LIN {X 0,Y 185.248,Z 515.043,A -85,B 0,C 180,E1 -23455.315,E2 -23455.315} C_VEL
LIN {X 0,Y 180.266,Z 523.701,A -85,B 0,C 180,E1 -23458.243,E2 -23458.243} C_VEL
LIN {X 0,Y 175.893,Z 530.639,A -85,B 0,C 180,E1 -23461.349,E2 -23461.349} C_VEL
LIN {X 0,Y 172.117,Z 536.223,A -85,B 0,C 180,E1 -23464.612,E2 -23464.612} C_VEL
LIN {X 0,Y 168.809,Z 540.646,A -85,B 0,C 180,E1 -23467.994,E2 -23467.994} C_VEL
LIN {X 0,Y 166.906,Z 542.994,A -85,B 0,C 180,E1 -23470.314,E2 -23470.314} C_VEL
LIN {X 0,Y 165.318,Z 544.923,A -85,B 0,C 180,E1 -23472.687,E2 -23472.687} C_VEL
LIN {X 0,Y 164.124,Z 546.443,A -85,B 0,C 180,E1 -23475.112,E2 -23475.112} C_VEL
LIN {X 0,Y 162.456,Z 548.229,A -85,B 0,C 180,E1 -23480.035,E2 -23480.035} C_VEL
LIN {X 0,Y 161.851,Z 548.504,A -85,B 0,C 180,E1 -23485.017,E2 -23485.017} C_VEL
LIN {X 0,Y 161.843,Z 548.032,A -85,B 0,C 180,E1 -23487.511,E2 -23487.511} C_VEL
LIN {X 0,Y 161.944,Z 547.156,A -85,B 0,C 180,E1 -23490,E2 -23490} C_VEL
LIN {X 0,Y 161.834,Z 545.704,A -85,B 0,C 180,E1 -23492.768,E2 -23492.768} C_VEL
LIN {X 0,Y 161.908,Z 543.109,A -85,B 0,C 180,E1 -23496.229,E2 -23496.229} C_VEL
LIN {X 0,Y 162.4,Z 539.305,A -85,B 0,C 180,E1 -23499.968,E2 -23499.968} C_VEL
LIN {X 0,Y 163.325,Z 534.348,A -85,B 0,C 180,E1 -23503.689,E2 -23503.689} C_VEL
LIN {X 0,Y 164.915,Z 528.1,A -85,B 0,C 180,E1 -23507.355,E2 -23507.355} C_VEL
LIN {X 0,Y 167.043,Z 520.275,A -85,B 0,C 180,E1 -23510.953,E2 -23510.953} C_VEL
LIN {X 0,Y 168.207,Z 515.825,A -85,B 0,C 180,E1 -23512.657,E2 -23512.657} C_VEL
LIN {X 0,Y 170.737,Z 506.615,A -85,B 0,C 180,E1 -23515.607,E2 -23515.607} C_VEL
LIN {X 0,Y 172.299,Z 500.233,A -85,B 0,C 180,E1 -23517.314,E2 -23517.314} C_VEL
LIN {X 0,Y 172.549,Z 488.695,A -85,B 0,C 180,E1 -23520.136,E2 -23520.136} C_VEL
LIN {X 0,Y 171.858,Z 483.921,A -85,B 0,C 180,E1 -23521.271,E2 -23521.271} C_VEL
LIN {X 0,Y 168.91,Z 476.415,A -85,B 0,C 180,E1 -23523.212,E2 -23523.212} C_VEL
LIN {X 0,Y 166.129,Z 470.335,A -85,B 0,C 180,E1 -23524.727,E2 -23524.727} C_VEL
LIN {X 0,Y 164.489,Z 465.427,A -85,B 0,C 180,E1 -23525.769,E2 -23525.769} C_VEL
LIN {X 0,Y 164.105,Z 463.69,A -85,B 0,C 180,E1 -23526.084,E2 -23526.084} C_VEL
LIN {X 0,Y 161.974,Z 452.52,A -85,B 0,C 180,E1 -23527.886,E2 -23527.886} C_VEL
LIN {X 0,Y 160.13,Z 446.258,A -85,B 0,C 180,E1 -23528.883,E2 -23528.883} C_VEL
LIN {X 0,Y 158.77,Z 443.265,A -85,B 0,C 180,E1 -23529.445,E2 -23529.445} C_VEL
LIN {X 0,Y 158.538,Z 442.036,A -85,B 0,C 180,E1 -23529.667,E2 -23529.667} C_VEL
LIN {X 0,Y 157.914,Z 438.937,A -85,B 0,C 180,E1 -23534.594,E2 -23534.594} C_VEL
LIN {X 0,Y 157.284,Z 435.898,A -85,B 0,C 180,E1 -23539.983,E2 -23539.983} C_VEL
LIN {X 0,Y 157.277,Z 435.896,A -85,B 0,C 180,E1 -23544.485,E2 -23544.485} C_VEL
LIN {X 0,Y 157.29,Z 435.892,A -85,B 0,C 180,E1 -23548.095,E2 -23548.095} C_VEL
LIN {X 0,Y 157.319,Z 435.868,A -85,B 0,C 180,E1 -23553.465,E2 -23553.465} C_VEL
LIN {X 0,Y 157.391,Z 435.873,A -85,B 0,C 180,E1 -23559.667,E2 -23559.667} C_VEL
LIN {X 0,Y 157.436,Z 435.841,A -85,B 0,C 180,E1 -23564.464,E2 -23564.464} C_VEL
LIN {X 0,Y 157.744,Z 435.835,A -85,B 0,C 180,E1 -23569.734,E2 -23569.734} C_VEL
LIN {X 0,Y 157.816,Z 435.818,A -85,B 0,C 180,E1 -23572.322,E2 -23572.322} C_VEL
LIN {X 0,Y 158.255,Z 435.755,A -85,B 0,C 180,E1 -23580,E2 -23580} C_VEL
LIN {X 0,Y 157.807,Z 435.813,A -85,B 0,C 180,E1 -23587.678,E2 -23587.678} C_VEL
LIN {X 0,Y 157.668,Z 435.803,A -85,B 0,C 180,E1 -23591.301,E2 -23591.301} C_VEL
LIN {X 0,Y 157.45,Z 435.863,A -85,B 0,C 180,E1 -23595.534,E2 -23595.534} C_VEL
LIN {X 0,Y 157.366,Z 435.877,A -85,B 0,C 180,E1 -23600.933,E2 -23600.933} C_VEL
LIN {X 0,Y 157.306,Z 435.888,A -85,B 0,C 180,E1 -23606.681,E2 -23606.681} C_VEL
LIN {X 0,Y 157.273,Z 435.894,A -85,B 0,C 180,E1 -23612.427,E2 -23612.427} C_VEL
LIN {X 0,Y 157.322,Z 435.881,A -85,B 0,C 180,E1 -23616.478,E2 -23616.478} C_VEL
LIN {X 0,Y 157.293,Z 435.891,A -85,B 0,C 180,E1 -23622.083,E2 -23622.083} C_VEL
LIN {X 0,Y 157.311,Z 435.889,A -85,B 0,C 180,E1 -23625.627,E2 -23625.627} C_VEL
LIN {X 0,Y 157.29,Z 435.892,A -85,B 0,C 180,E1 -23631.279,E2 -23631.279} C_VEL
LIN {X 0,Y 157.293,Z 435.89,A -85,B 0,C 180,E1 -23634.491,E2 -23634.491} C_VEL
LIN {X 0,Y 157.293,Z 435.892,A -85,B 0,C 180,E1 -23638.096,E2 -23638.096} C_VEL
LIN {X 0,Y 157.413,Z 436.05,A -85,B 0,C 180,E1 -23644.324,E2 -23644.324} C_VEL
LIN {X 0,Y 158.472,Z 438.848,A -85,B 0,C 180,E1 -23644.818,E2 -23644.818} C_VEL
LIN {X 0,Y 159.937,Z 441.308,A -85,B 0,C 180,E1 -23645.373,E2 -23645.373} C_VEL
LIN {X 0,Y 162.244,Z 447.436,A -85,B 0,C 180,E1 -23646.537,E2 -23646.537} C_VEL
LIN {X 0,Y 165.121,Z 458.356,A -85,B 0,C 180,E1 -23648.593,E2 -23648.593} C_VEL
LIN {X 0,Y 166.934,Z 469.095,A -85,B 0,C 180,E1 -23650.769,E2 -23650.769} C_VEL
LIN {X 0,Y 167.973,Z 478.773,A -85,B 0,C 180,E1 -23652.97,E2 -23652.97} C_VEL
LIN {X 0,Y 168.048,Z 485.349,A -85,B 0,C 180,E1 -23654.587,E2 -23654.587} C_VEL
LIN {X 0,Y 165.391,Z 495.531,A -85,B 0,C 180,E1 -23657.11,E2 -23657.11} C_VEL
LIN {X 0,Y 162.736,Z 504.865,A -85,B 0,C 180,E1 -23660.053,E2 -23660.053} C_VEL
LIN {X 0,Y 160.012,Z 513.909,A -85,B 0,C 180,E1 -23663.697,E2 -23663.697} C_VEL
LIN {X 0,Y 157.857,Z 521.199,A -85,B 0,C 180,E1 -23667.449,E2 -23667.449} C_VEL
LIN {X 0,Y 156.377,Z 527.011,A -85,B 0,C 180,E1 -23671.288,E2 -23671.288} C_VEL
LIN {X 0,Y 155.326,Z 531.874,A -85,B 0,C 180,E1 -23675.485,E2 -23675.485} C_VEL
LIN {X 0,Y 154.858,Z 534.018,A -85,B 0,C 180,E1 -23677.826,E2 -23677.826} C_VEL
LIN {X 0,Y 154.489,Z 536.015,A -85,B 0,C 180,E1 -23680.485,E2 -23680.485} C_VEL
LIN {X 0,Y 154.366,Z 537.581,A -85,B 0,C 180,E1 -23683.158,E2 -23683.158} C_VEL
LIN {X 0,Y 154.602,Z 539.136,A -85,B 0,C 180,E1 -23687.327,E2 -23687.327} C_VEL
LIN {X 0,Y 155.216,Z 539.674,A -85,B 0,C 180,E1 -23691.237,E2 -23691.237} C_VEL
LIN {X 0,Y 156.841,Z 539.037,A -85,B 0,C 180,E1 -23696.339,E2 -23696.339} C_VEL
LIN {X 0,Y 158.206,Z 537.971,A -85,B 0,C 180,E1 -23699.252,E2 -23699.252} C_VEL
LIN {X 0,Y 159.765,Z 536.553,A -85,B 0,C 180,E1 -23701.862,E2 -23701.862} C_VEL
LIN {X 0,Y 162.668,Z 533.529,A -85,B 0,C 180,E1 -23705.68,E2 -23705.68} C_VEL
LIN {X 0,Y 166.199,Z 529.371,A -85,B 0,C 180,E1 -23709.368,E2 -23709.368} C_VEL
LIN {X 0,Y 170.381,Z 523.946,A -85,B 0,C 180,E1 -23712.89,E2 -23712.89} C_VEL
LIN {X 0,Y 175.179,Z 517.076,A -85,B 0,C 180,E1 -23716.231,E2 -23716.231} C_VEL
LIN {X 0,Y 180.487,Z 508.46,A -85,B 0,C 180,E1 -23719.403,E2 -23719.403} C_VEL
LIN {X 0,Y 182.402,Z 505.098,A -85,B 0,C 180,E1 -23720.408,E2 -23720.408} C_VEL
LIN {X 0,Y 183.047,Z 501.795,A -85,B 0,C 180,E1 -23721.655,E2 -23721.655} C_VEL
LIN {X 0,Y 183.419,Z 493.353,A -85,B 0,C 180,E1 -23724.918,E2 -23724.918} C_VEL
LIN {X 0,Y 182.864,Z 486.054,A -85,B 0,C 180,E1 -23727.727,E2 -23727.727} C_VEL
LIN {X 0,Y 181.46,Z 479.589,A -85,B 0,C 180,E1 -23730.426,E2 -23730.426} C_VEL
LIN {X 0,Y 178.98,Z 472.271,A -85,B 0,C 180,E1 -23733.785,E2 -23733.785} C_VEL
LIN {X 0,Y 177.584,Z 468.714,A -85,B 0,C 180,E1 -23735.537,E2 -23735.537} C_VEL
LIN {X 0,Y 175.789,Z 464.643,A -85,B 0,C 180,E1 -23737.679,E2 -23737.679} C_VEL
LIN {X 0,Y 172.805,Z 459.443,A -85,B 0,C 180,E1 -23741.013,E2 -23741.013} C_VEL
LIN {X 0,Y 170.994,Z 455.9,A -85,B 0,C 180,E1 -23743.28,E2 -23743.28} C_VEL
LIN {X 0,Y 168.006,Z 451.559,A -85,B 0,C 180,E1 -23747.007,E2 -23747.007} C_VEL
LIN {X 0,Y 167.308,Z 449.863,A -85,B 0,C 180,E1 -23748.184,E2 -23748.184} C_VEL
LIN {X 0,Y 164.416,Z 446.661,A -85,B 0,C 180,E1 -23752.478,E2 -23752.478} C_VEL
LIN {X 0,Y 163.46,Z 444.35,A -85,B 0,C 180,E1 -23754.758,E2 -23754.758} C_VEL
LIN {X 0,Y 161.309,Z 442.705,A -85,B 0,C 180,E1 -23760,E2 -23760} C_VEL
LIN {X 0,Y 160.22,Z 442.45,A -85,B 0,C 180,E1 -23767.562,E2 -23767.562} C_VEL
LIN {X 0,Y 160.844,Z 443.769,A -85,B 0,C 180,E1 -23772.62,E2 -23772.62} C_VEL
LIN {X 0,Y 163.558,Z 446.46,A -85,B 0,C 180,E1 -23779.484,E2 -23779.484} C_VEL
LIN {X 0,Y 164.954,Z 450.06,A -85,B 0,C 180,E1 -23782.548,E2 -23782.548} C_VEL
LIN {X 0,Y 167.772,Z 453.476,A -85,B 0,C 180,E1 -23786.429,E2 -23786.429} C_VEL
LIN {X 0,Y 169.173,Z 456.816,A -85,B 0,C 180,E1 -23788.539,E2 -23788.539} C_VEL
LIN {X 0,Y 171.221,Z 459.675,A -85,B 0,C 180,E1 -23790.868,E2 -23790.868} C_VEL
LIN {X 0,Y 172.912,Z 463.461,A -85,B 0,C 180,E1 -23792.999,E2 -23792.999} C_VEL
LIN {X 0,Y 174.138,Z 465.815,A -85,B 0,C 180,E1 -23794.404,E2 -23794.404} C_VEL
LIN {X 0,Y 176.569,Z 471.344,A -85,B 0,C 180,E1 -23797.245,E2 -23797.245} C_VEL
LIN {X 0,Y 179.659,Z 479.366,A -85,B 0,C 180,E1 -23800.938,E2 -23800.938} C_VEL
LIN {X 0,Y 181.699,Z 487.258,A -85,B 0,C 180,E1 -23804.126,E2 -23804.126} C_VEL
LIN {X 0,Y 182.158,Z 491.421,A -85,B 0,C 180,E1 -23805.602,E2 -23805.602} C_VEL
LIN {X 0,Y 182.082,Z 499.048,A -85,B 0,C 180,E1 -23808.149,E2 -23808.149} C_VEL
LIN {X 0,Y 180.895,Z 508.937,A -85,B 0,C 180,E1 -23811.566,E2 -23811.566} C_VEL
LIN {X 0,Y 179.382,Z 515.508,A -85,B 0,C 180,E1 -23814.007,E2 -23814.007} C_VEL
LIN {X 0,Y 175.101,Z 522.707,A -85,B 0,C 180,E1 -23816.504,E2 -23816.504} C_VEL
LIN {X 0,Y 170.424,Z 529.828,A -85,B 0,C 180,E1 -23819.658,E2 -23819.658} C_VEL
LIN {X 0,Y 165.735,Z 536.348,A -85,B 0,C 180,E1 -23823.561,E2 -23823.561} C_VEL
LIN {X 0,Y 162.222,Z 540.694,A -85,B 0,C 180,E1 -23827.051,E2 -23827.051} C_VEL
LIN {X 0,Y 158.529,Z 544.901,A -85,B 0,C 180,E1 -23831.921,E2 -23831.921} C_VEL
LIN {X 0,Y 157.231,Z 546.355,A -85,B 0,C 180,E1 -23834.443,E2 -23834.443} C_VEL
LIN {X 0,Y 155.456,Z 548.072,A -85,B 0,C 180,E1 -23839.581,E2 -23839.581} C_VEL
LIN {X 0,Y 154.76,Z 548.267,A -85,B 0,C 180,E1 -23844.789,E2 -23844.789} C_VEL
LIN {X 0,Y 154.758,Z 547.701,A -85,B 0,C 180,E1 -23847.558,E2 -23847.558} C_VEL
LIN {X 0,Y 154.854,Z 546.841,A -85,B 0,C 180,E1 -23849.999,E2 -23849.999} C_VEL
LIN {X 0,Y 154.742,Z 545.519,A -85,B 0,C 180,E1 -23852.603,E2 -23852.603} C_VEL
LIN {X 0,Y 154.855,Z 542.694,A -85,B 0,C 180,E1 -23856.514,E2 -23856.514} C_VEL
LIN {X 0,Y 155.4,Z 538.819,A -85,B 0,C 180,E1 -23860.421,E2 -23860.421} C_VEL
LIN {X 0,Y 156.397,Z 533.783,A -85,B 0,C 180,E1 -23864.308,E2 -23864.308} C_VEL
LIN {X 0,Y 158.11,Z 527.447,A -85,B 0,C 180,E1 -23868.128,E2 -23868.128} C_VEL
LIN {X 0,Y 160.414,Z 519.48,A -85,B 0,C 180,E1 -23871.863,E2 -23871.863} C_VEL
LIN {X 0,Y 162.42,Z 512.051,A -85,B 0,C 180,E1 -23874.675,E2 -23874.675} C_VEL
LIN {X 0,Y 165.153,Z 502.458,A -85,B 0,C 180,E1 -23877.565,E2 -23877.565} C_VEL
LIN {X 0,Y 165.664,Z 497.782,A -85,B 0,C 180,E1 -23878.852,E2 -23878.852} C_VEL
LIN {X 0,Y 165.875,Z 487.286,A -85,B 0,C 180,E1 -23881.466,E2 -23881.466} C_VEL
LIN {X 0,Y 165.536,Z 476.278,A -85,B 0,C 180,E1 -23883.79,E2 -23883.79} C_VEL
LIN {X 0,Y 164.288,Z 464.832,A -85,B 0,C 180,E1 -23885.892,E2 -23885.892} C_VEL
LIN {X 0,Y 164.105,Z 463.69,A -85,B 0,C 180,E1 -23886.084,E2 -23886.084} C_VEL
LIN {X 0,Y 162.955,Z 460.45,A -85,B 0,C 180,E1 -23886.762,E2 -23886.762} C_VEL
LIN {X 0,Y 159.595,Z 455.978,A -85,B 0,C 180,E1 -23888.04,E2 -23888.04} C_VEL
LIN {X 0,Y 155.141,Z 450.752,A -85,B 0,C 180,E1 -23889.646,E2 -23889.646} C_VEL
LIN {X 0,Y 153.972,Z 448.703,A -85,B 0,C 180,E1 -23890.138,E2 -23890.138} C_VEL
LIN {X 0,Y 152.57,Z 445.411,A -85,B 0,C 180,E1 -23890.784,E2 -23890.784} C_VEL
LIN {X 0,Y 151.417,Z 442.505,A -85,B 0,C 180,E1 -23891.333,E2 -23891.333} C_VEL
LIN {X 0,Y 151.297,Z 441.796,A -85,B 0,C 180,E1 -23891.519,E2 -23891.519} C_VEL
LIN {X 0,Y 150.741,Z 439.381,A -85,B 0,C 180,E1 -23895.625,E2 -23895.625} C_VEL
LIN {X 0,Y 150.224,Z 436.778,A -85,B 0,C 180,E1 -23900.399,E2 -23900.399} C_VEL
LIN {X 0,Y 150.188,Z 436.777,A -85,B 0,C 180,E1 -23905.837,E2 -23905.837} C_VEL
LIN {X 0,Y 150.204,Z 436.771,A -85,B 0,C 180,E1 -23909.023,E2 -23909.023} C_VEL
LIN {X 0,Y 150.241,Z 436.745,A -85,B 0,C 180,E1 -23912.717,E2 -23912.717} C_VEL
LIN {X 0,Y 150.348,Z 436.752,A -85,B 0,C 180,E1 -23919.207,E2 -23919.207} C_VEL
LIN {X 0,Y 150.346,Z 436.72,A -85,B 0,C 180,E1 -23923.711,E2 -23923.711} C_VEL
LIN {X 0,Y 150.658,Z 436.718,A -85,B 0,C 180,E1 -23929.245,E2 -23929.245} C_VEL
LIN {X 0,Y 150.752,Z 436.701,A -85,B 0,C 180,E1 -23931.96,E2 -23931.96} C_VEL
LIN {X 0,Y 151.215,Z 436.631,A -85,B 0,C 180,E1 -23940,E2 -23940} C_VEL
LIN {X 0,Y 150.741,Z 436.689,A -85,B 0,C 180,E1 -23948.04,E2 -23948.04} C_VEL
LIN {X 0,Y 150.602,Z 436.681,A -85,B 0,C 180,E1 -23951.491,E2 -23951.491} C_VEL
LIN {X 0,Y 150.358,Z 436.749,A -85,B 0,C 180,E1 -23956.287,E2 -23956.287} C_VEL
LIN {X 0,Y 150.347,Z 436.752,A -85,B 0,C 180,E1 -23960.792,E2 -23960.792} C_VEL
LIN {X 0,Y 150.238,Z 436.767,A -85,B 0,C 180,E1 -23967.28,E2 -23967.28} C_VEL
LIN {X 0,Y 150.214,Z 436.773,A -85,B 0,C 180,E1 -23972.634,E2 -23972.634} C_VEL
LIN {X 0,Y 150.233,Z 436.767,A -85,B 0,C 180,E1 -23977.455,E2 -23977.455} C_VEL
LIN {X 0,Y 150.234,Z 436.771,A -85,B 0,C 180,E1 -23981.543,E2 -23981.543} C_VEL
LIN {X 0,Y 150.286,Z 436.764,A -85,B 0,C 180,E1 -23985.458,E2 -23985.458} C_VEL
LIN {X 0,Y 150.236,Z 436.769,A -85,B 0,C 180,E1 -23989.088,E2 -23989.088} C_VEL
LIN {X 0,Y 150.238,Z 436.77,A -85,B 0,C 180,E1 -23992.678,E2 -23992.678} C_VEL
LIN {X 0,Y 150.217,Z 436.773,A -85,B 0,C 180,E1 -23997.366,E2 -23997.366} C_VEL
LIN {X 0,Y 150.243,Z 436.771,A -85,B 0,C 180,E1 -24002.494,E2 -24002.494} C_VEL
LIN {X 0,Y 151.372,Z 439.8,A -85,B 0,C 180,E1 -24003.108,E2 -24003.108} C_VEL
LIN {X 0,Y 152.628,Z 441.712,A -85,B 0,C 180,E1 -24003.616,E2 -24003.616} C_VEL
LIN {X 0,Y 155.281,Z 446.867,A -85,B 0,C 180,E1 -24004.849,E2 -24004.849} C_VEL
LIN {X 0,Y 158.629,Z 458.919,A -85,B 0,C 180,E1 -24007.306,E2 -24007.306} C_VEL
LIN {X 0,Y 160.475,Z 470.171,A -85,B 0,C 180,E1 -24009.74,E2 -24009.74} C_VEL
LIN {X 0,Y 161.422,Z 480.564,A -85,B 0,C 180,E1 -24012.257,E2 -24012.257} C_VEL
LIN {X 0,Y 161.347,Z 486.487,A -85,B 0,C 180,E1 -24013.788,E2 -24013.788} C_VEL
LIN {X 0,Y 158.431,Z 496.914,A -85,B 0,C 180,E1 -24016.533,E2 -24016.533} C_VEL
LIN {X 0,Y 155.735,Z 506.012,A -85,B 0,C 180,E1 -24019.601,E2 -24019.601} C_VEL
LIN {X 0,Y 152.913,Z 514.903,A -85,B 0,C 180,E1 -24023.403,E2 -24023.403} C_VEL
LIN {X 0,Y 150.734,Z 522.021,A -85,B 0,C 180,E1 -24027.328,E2 -24027.328} C_VEL
LIN {X 0,Y 149.214,Z 527.691,A -85,B 0,C 180,E1 -24031.35,E2 -24031.35} C_VEL
LIN {X 0,Y 148.217,Z 532.161,A -85,B 0,C 180,E1 -24035.442,E2 -24035.442} C_VEL
LIN {X 0,Y 147.691,Z 534.539,A -85,B 0,C 180,E1 -24038.208,E2 -24038.208} C_VEL
LIN {X 0,Y 147.363,Z 536.487,A -85,B 0,C 180,E1 -24040.998,E2 -24040.998} C_VEL
LIN {X 0,Y 147.266,Z 537.961,A -85,B 0,C 180,E1 -24043.805,E2 -24043.805} C_VEL
LIN {X 0,Y 147.531,Z 539.324,A -85,B 0,C 180,E1 -24047.685,E2 -24047.685} C_VEL
LIN {X 0,Y 148.331,Z 539.896,A -85,B 0,C 180,E1 -24052.275,E2 -24052.275} C_VEL
LIN {X 0,Y 150.007,Z 539.268,A -85,B 0,C 180,E1 -24057.106,E2 -24057.106} C_VEL
LIN {X 0,Y 151.742,Z 538.013,A -85,B 0,C 180,E1 -24060.628,E2 -24060.628} C_VEL
LIN {X 0,Y 154.935,Z 535.114,A -85,B 0,C 180,E1 -24065.265,E2 -24065.265} C_VEL
LIN {X 0,Y 159.14,Z 530.647,A -85,B 0,C 180,E1 -24069.818,E2 -24069.818} C_VEL
LIN {X 0,Y 164.205,Z 524.591,A -85,B 0,C 180,E1 -24074.067,E2 -24074.067} C_VEL
LIN {X 0,Y 169.231,Z 517.827,A -85,B 0,C 180,E1 -24077.488,E2 -24077.488} C_VEL
LIN {X 0,Y 174.767,Z 509.35,A -85,B 0,C 180,E1 -24080.724,E2 -24080.724} C_VEL
LIN {X 0,Y 176.697,Z 506.03,A -85,B 0,C 180,E1 -24081.77,E2 -24081.77} C_VEL
LIN {X 0,Y 177.431,Z 500.168,A -85,B 0,C 180,E1 -24084.251,E2 -24084.251} C_VEL
LIN {X 0,Y 177.621,Z 492.175,A -85,B 0,C 180,E1 -24087.539,E2 -24087.539} C_VEL
LIN {X 0,Y 176.823,Z 486.029,A -85,B 0,C 180,E1 -24090.212,E2 -24090.212} C_VEL
LIN {X 0,Y 174.92,Z 478.606,A -85,B 0,C 180,E1 -24093.771,E2 -24093.771} C_VEL
LIN {X 0,Y 173.381,Z 474.2,A -85,B 0,C 180,E1 -24096.087,E2 -24096.087} C_VEL
LIN {X 0,Y 171.778,Z 470.128,A -85,B 0,C 180,E1 -24098.395,E2 -24098.395} C_VEL
LIN {X 0,Y 169.164,Z 465.061,A -85,B 0,C 180,E1 -24101.845,E2 -24101.845} C_VEL
LIN {X 0,Y 167.59,Z 461.677,A -85,B 0,C 180,E1 -24104.182,E2 -24104.182} C_VEL
LIN {X 0,Y 165.182,Z 457.75,A -85,B 0,C 180,E1 -24107.718,E2 -24107.718} C_VEL
LIN {X 0,Y 164.566,Z 456.199,A -85,B 0,C 180,E1 -24108.92,E2 -24108.92} C_VEL
LIN {X 0,Y 162.033,Z 452.791,A -85,B 0,C 180,E1 -24113.463,E2 -24113.463} C_VEL
LIN {X 0,Y 161.402,Z 451.058,A -85,B 0,C 180,E1 -24115.317,E2 -24115.317} C_VEL
LIN {X 0,Y 159.36,Z 449.483,A -85,B 0,C 180,E1 -24121.264,E2 -24121.264} C_VEL
LIN {X 0,Y 158.693,Z 449.486,A -85,B 0,C 180,E1 -24128.276,E2 -24128.276} C_VEL
LIN {X 0,Y 159.836,Z 451.546,A -85,B 0,C 180,E1 -24134.906,E2 -24134.906} C_VEL
LIN {X 0,Y 161.452,Z 453.152,A -85,B 0,C 180,E1 -24138.909,E2 -24138.909} C_VEL
LIN {X 0,Y 162.813,Z 456.916,A -85,B 0,C 180,E1 -24142.359,E2 -24142.359} C_VEL
LIN {X 0,Y 164.678,Z 459.264,A -85,B 0,C 180,E1 -24145.263,E2 -24145.263} C_VEL
LIN {X 0,Y 166.97,Z 464.198,A -85,B 0,C 180,E1 -24148.951,E2 -24148.951} C_VEL
LIN {X 0,Y 168.1,Z 466.338,A -85,B 0,C 180,E1 -24150.527,E2 -24150.527} C_VEL
LIN {X 0,Y 170.523,Z 471.909,A -85,B 0,C 180,E1 -24153.95,E2 -24153.95} C_VEL
LIN {X 0,Y 173.072,Z 478.552,A -85,B 0,C 180,E1 -24157.526,E2 -24157.526} C_VEL
LIN {X 0,Y 175.119,Z 485.035,A -85,B 0,C 180,E1 -24160.628,E2 -24160.628} C_VEL
LIN {X 0,Y 176.514,Z 491.858,A -85,B 0,C 180,E1 -24163.574,E2 -24163.574} C_VEL
LIN {X 0,Y 176.54,Z 498.862,A -85,B 0,C 180,E1 -24166.136,E2 -24166.136} C_VEL
LIN {X 0,Y 175.511,Z 507.179,A -85,B 0,C 180,E1 -24169.149,E2 -24169.149} C_VEL
LIN {X 0,Y 173.991,Z 514.433,A -85,B 0,C 180,E1 -24171.976,E2 -24171.976} C_VEL
LIN {X 0,Y 172.876,Z 517.473,A -85,B 0,C 180,E1 -24173.156,E2 -24173.156} C_VEL
LIN {X 0,Y 167.532,Z 525.542,A -85,B 0,C 180,E1 -24176.232,E2 -24176.232} C_VEL
LIN {X 0,Y 162.444,Z 532.614,A -85,B 0,C 180,E1 -24179.851,E2 -24179.851} C_VEL
LIN {X 0,Y 158.083,Z 538.031,A -85,B 0,C 180,E1 -24183.604,E2 -24183.604} C_VEL
LIN {X 0,Y 154.624,Z 541.949,A -85,B 0,C 180,E1 -24187.273,E2 -24187.273} C_VEL
LIN {X 0,Y 151.777,Z 544.865,A -85,B 0,C 180,E1 -24191.087,E2 -24191.087} C_VEL
LIN {X 0,Y 149.267,Z 547.279,A -85,B 0,C 180,E1 -24196.384,E2 -24196.384} C_VEL
LIN {X 0,Y 147.945,Z 548.175,A -85,B 0,C 180,E1 -24201.806,E2 -24201.806} C_VEL
LIN {X 0,Y 147.691,Z 548.014,A -85,B 0,C 180,E1 -24204.538,E2 -24204.538} C_VEL
LIN {X 0,Y 147.677,Z 547.252,A -85,B 0,C 180,E1 -24208.022,E2 -24208.022} C_VEL
LIN {X 0,Y 147.767,Z 546.522,A -85,B 0,C 180,E1 -24209.999,E2 -24209.999} C_VEL
LIN {X 0,Y 147.646,Z 545.166,A -85,B 0,C 180,E1 -24212.728,E2 -24212.728} C_VEL
LIN {X 0,Y 147.783,Z 542.271,A -85,B 0,C 180,E1 -24216.827,E2 -24216.827} C_VEL
LIN {X 0,Y 148.381,Z 538.321,A -85,B 0,C 180,E1 -24220.92,E2 -24220.92} C_VEL
LIN {X 0,Y 149.695,Z 532.204,A -85,B 0,C 180,E1 -24225.661,E2 -24225.661} C_VEL
LIN {X 0,Y 151.707,Z 525.503,A -85,B 0,C 180,E1 -24229.624,E2 -24229.624} C_VEL
LIN {X 0,Y 154.255,Z 517.157,A -85,B 0,C 180,E1 -24233.493,E2 -24233.493} C_VEL
LIN {X 0,Y 155.362,Z 512.973,A -85,B 0,C 180,E1 -24235.127,E2 -24235.127} C_VEL
LIN {X 0,Y 158.222,Z 503.532,A -85,B 0,C 180,E1 -24238.16,E2 -24238.16} C_VEL
LIN {X 0,Y 158.913,Z 499.006,A -85,B 0,C 180,E1 -24239.471,E2 -24239.471} C_VEL
LIN {X 0,Y 159.278,Z 487.857,A -85,B 0,C 180,E1 -24242.418,E2 -24242.418} C_VEL
LIN {X 0,Y 159.086,Z 477.591,A -85,B 0,C 180,E1 -24244.722,E2 -24244.722} C_VEL
LIN {X 0,Y 157.935,Z 465.896,A -85,B 0,C 180,E1 -24247.04,E2 -24247.04} C_VEL
LIN {X 0,Y 155.889,Z 454.167,A -85,B 0,C 180,E1 -24249.093,E2 -24249.093} C_VEL
LIN {X 0,Y 153.972,Z 448.703,A -85,B 0,C 180,E1 -24250.138,E2 -24250.138} C_VEL
LIN {X 0,Y 151.998,Z 445.869,A -85,B 0,C 180,E1 -24250.948,E2 -24250.948} C_VEL
LIN {X 0,Y 149.545,Z 443.812,A -85,B 0,C 180,E1 -24251.936,E2 -24251.936} C_VEL
LIN {X 0,Y 146.327,Z 441.924,A -85,B 0,C 180,E1 -24253.517,E2 -24253.517} C_VEL
LIN {X 0,Y 144.037,Z 440.581,A -85,B 0,C 180,E1 -24255.418,E2 -24255.418} C_VEL
LIN {X 0,Y 143.604,Z 439.995,A -85,B 0,C 180,E1 -24256.468,E2 -24256.468} C_VEL
LIN {X 0,Y 143.148,Z 437.659,A -85,B 0,C 180,E1 -24261.182,E2 -24261.182} C_VEL
LIN {X 0,Y 143.179,Z 437.651,A -85,B 0,C 180,E1 -24267.32,E2 -24267.32} C_VEL
LIN {X 0,Y 143.187,Z 437.623,A -85,B 0,C 180,E1 -24272.062,E2 -24272.062} C_VEL
LIN {X 0,Y 143.274,Z 437.634,A -85,B 0,C 180,E1 -24278.745,E2 -24278.745} C_VEL
LIN {X 0,Y 143.29,Z 437.598,A -85,B 0,C 180,E1 -24282.885,E2 -24282.885} C_VEL
LIN {X 0,Y 143.591,Z 437.597,A -85,B 0,C 180,E1 -24288.709,E2 -24288.709} C_VEL
LIN {X 0,Y 143.67,Z 437.586,A -85,B 0,C 180,E1 -24291.561,E2 -24291.561} C_VEL
LIN {X 0,Y 144.174,Z 437.506,A -85,B 0,C 180,E1 -24300,E2 -24300} C_VEL
LIN {X 0,Y 143.659,Z 437.566,A -85,B 0,C 180,E1 -24308.439,E2 -24308.439} C_VEL
LIN {X 0,Y 143.544,Z 437.559,A -85,B 0,C 180,E1 -24311.712,E2 -24311.712} C_VEL
LIN {X 0,Y 143.297,Z 437.633,A -85,B 0,C 180,E1 -24317.113,E2 -24317.113} C_VEL
LIN {X 0,Y 143.273,Z 437.63,A -85,B 0,C 180,E1 -24321.254,E2 -24321.254} C_VEL
LIN {X 0,Y 143.184,Z 437.641,A -85,B 0,C 180,E1 -24327.935,E2 -24327.935} C_VEL
LIN {X 0,Y 143.166,Z 437.65,A -85,B 0,C 180,E1 -24333.436,E2 -24333.436} C_VEL
LIN {X 0,Y 143.127,Z 437.655,A -85,B 0,C 180,E1 -24339.668,E2 -24339.668} C_VEL
LIN {X 0,Y 143.18,Z 437.648,A -85,B 0,C 180,E1 -24343.408,E2 -24343.408} C_VEL
LIN {X 0,Y 143.169,Z 437.651,A -85,B 0,C 180,E1 -24347.419,E2 -24347.419} C_VEL
LIN {X 0,Y 143.167,Z 437.65,A -85,B 0,C 180,E1 -24351.76,E2 -24351.76} C_VEL
LIN {X 0,Y 143.185,Z 437.649,A -85,B 0,C 180,E1 -24357.323,E2 -24357.323} C_VEL
LIN {X 0,Y 143.144,Z 437.774,A -85,B 0,C 180,E1 -24360.553,E2 -24360.553} C_VEL
LIN {X 0,Y 144.243,Z 440.681,A -85,B 0,C 180,E1 -24361.173,E2 -24361.173} C_VEL
LIN {X 0,Y 145.618,Z 442.737,A -85,B 0,C 180,E1 -24361.801,E2 -24361.801} C_VEL
LIN {X 0,Y 149.699,Z 450.427,A -85,B 0,C 180,E1 -24363.896,E2 -24363.896} C_VEL
LIN {X 0,Y 152.533,Z 461.393,A -85,B 0,C 180,E1 -24366.334,E2 -24366.334} C_VEL
LIN {X 0,Y 154.188,Z 472.769,A -85,B 0,C 180,E1 -24368.98,E2 -24368.98} C_VEL
LIN {X 0,Y 154.908,Z 482.352,A -85,B 0,C 180,E1 -24371.484,E2 -24371.484} C_VEL
LIN {X 0,Y 154.835,Z 487.061,A -85,B 0,C 180,E1 -24372.791,E2 -24372.791} C_VEL
LIN {X 0,Y 152.164,Z 496.271,A -85,B 0,C 180,E1 -24375.285,E2 -24375.285} C_VEL
LIN {X 0,Y 149.251,Z 505.528,A -85,B 0,C 180,E1 -24378.456,E2 -24378.456} C_VEL
LIN {X 0,Y 146.272,Z 514.53,A -85,B 0,C 180,E1 -24382.408,E2 -24382.408} C_VEL
LIN {X 0,Y 143.935,Z 521.778,A -85,B 0,C 180,E1 -24386.501,E2 -24386.501} C_VEL
LIN {X 0,Y 142.526,Z 526.659,A -85,B 0,C 180,E1 -24390.001,E2 -24390.001} C_VEL
LIN {X 0,Y 141.401,Z 531.175,A -85,B 0,C 180,E1 -24394.043,E2 -24394.043} C_VEL
LIN {X 0,Y 140.508,Z 535.063,A -85,B 0,C 180,E1 -24398.631,E2 -24398.631} C_VEL
LIN {X 0,Y 140.214,Z 536.935,A -85,B 0,C 180,E1 -24401.566,E2 -24401.566} C_VEL
LIN {X 0,Y 140.195,Z 538.337,A -85,B 0,C 180,E1 -24404.516,E2 -24404.516} C_VEL
LIN {X 0,Y 140.479,Z 539.513,A -85,B 0,C 180,E1 -24408.096,E2 -24408.096} C_VEL
LIN {X 0,Y 141.494,Z 540.086,A -85,B 0,C 180,E1 -24413.413,E2 -24413.413} C_VEL
LIN {X 0,Y 143.185,Z 539.505,A -85,B 0,C 180,E1 -24417.934,E2 -24417.934} C_VEL
LIN {X 0,Y 145.384,Z 538.028,A -85,B 0,C 180,E1 -24422.124,E2 -24422.124} C_VEL
LIN {X 0,Y 148.486,Z 535.408,A -85,B 0,C 180,E1 -24426.427,E2 -24426.427} C_VEL
LIN {X 0,Y 152.089,Z 531.904,A -85,B 0,C 180,E1 -24430.311,E2 -24430.311} C_VEL
LIN {X 0,Y 156.393,Z 527.232,A -85,B 0,C 180,E1 -24434.028,E2 -24434.028} C_VEL
LIN {X 0,Y 161.541,Z 520.961,A -85,B 0,C 180,E1 -24437.697,E2 -24437.697} C_VEL
LIN {X 0,Y 166.522,Z 514.126,A -85,B 0,C 180,E1 -24440.724,E2 -24440.724} C_VEL
LIN {X 0,Y 170.185,Z 508.666,A -85,B 0,C 180,E1 -24442.65,E2 -24442.65} C_VEL
LIN {X 0,Y 170.877,Z 506.927,A -85,B 0,C 180,E1 -24443.322,E2 -24443.322} C_VEL
LIN {X 0,Y 171.781,Z 500.013,A -85,B 0,C 180,E1 -24446.446,E2 -24446.446} C_VEL
LIN {X 0,Y 171.916,Z 493.981,A -85,B 0,C 180,E1 -24449.146,E2 -24449.146} C_VEL
LIN {X 0,Y 171.25,Z 488.417,A -85,B 0,C 180,E1 -24451.839,E2 -24451.839} C_VEL
LIN {X 0,Y 169.854,Z 482.595,A -85,B 0,C 180,E1 -24454.906,E2 -24454.906} C_VEL
LIN {X 0,Y 168.578,Z 478.569,A -85,B 0,C 180,E1 -24457.253,E2 -24457.253} C_VEL
LIN {X 0,Y 167.577,Z 475.464,A -85,B 0,C 180,E1 -24459.116,E2 -24459.116} C_VEL
LIN {X 0,Y 165.329,Z 470.535,A -85,B 0,C 180,E1 -24462.689,E2 -24462.689} C_VEL
LIN {X 0,Y 163.965,Z 467.36,A -85,B 0,C 180,E1 -24465.098,E2 -24465.098} C_VEL
LIN {X 0,Y 161.349,Z 462.252,A -85,B 0,C 180,E1 -24469.967,E2 -24469.967} C_VEL
LIN {X 0,Y 159.637,Z 459.567,A -85,B 0,C 180,E1 -24473.682,E2 -24473.682} C_VEL
LIN {X 0,Y 159.285,Z 458.378,A -85,B 0,C 180,E1 -24474.938,E2 -24474.938} C_VEL
LIN {X 0,Y 157.684,Z 456.449,A -85,B 0,C 180,E1 -24480,E2 -24480} C_VEL
LIN {X 0,Y 156.781,Z 456.138,A -85,B 0,C 180,E1 -24485.144,E2 -24485.144} C_VEL
LIN {X 0,Y 156.848,Z 456.591,A -85,B 0,C 180,E1 -24489.681,E2 -24489.681} C_VEL
LIN {X 0,Y 158.917,Z 459.496,A -85,B 0,C 180,E1 -24498.034,E2 -24498.034} C_VEL
LIN {X 0,Y 160.151,Z 463.362,A -85,B 0,C 180,E1 -24501.902,E2 -24501.902} C_VEL
LIN {X 0,Y 161.553,Z 465.287,A -85,B 0,C 180,E1 -24504.41,E2 -24504.41} C_VEL
LIN {X 0,Y 164.329,Z 471.511,A -85,B 0,C 180,E1 -24509.462,E2 -24509.462} C_VEL
LIN {X 0,Y 166.509,Z 477.414,A -85,B 0,C 180,E1 -24513.279,E2 -24513.279} C_VEL
LIN {X 0,Y 168.746,Z 484.184,A -85,B 0,C 180,E1 -24517.152,E2 -24517.152} C_VEL
LIN {X 0,Y 170.337,Z 490.674,A -85,B 0,C 180,E1 -24520.428,E2 -24520.428} C_VEL
LIN {X 0,Y 171.087,Z 495.532,A -85,B 0,C 180,E1 -24522.671,E2 -24522.671} C_VEL
LIN {X 0,Y 170.835,Z 501.465,A -85,B 0,C 180,E1 -24525.021,E2 -24525.021} C_VEL
LIN {X 0,Y 169.467,Z 509.814,A -85,B 0,C 180,E1 -24528.287,E2 -24528.287} C_VEL
LIN {X 0,Y 167.739,Z 516.468,A -85,B 0,C 180,E1 -24531.062,E2 -24531.062} C_VEL
LIN {X 0,Y 166.342,Z 519.376,A -85,B 0,C 180,E1 -24532.221,E2 -24532.221} C_VEL
LIN {X 0,Y 160.802,Z 527.03,A -85,B 0,C 180,E1 -24535.377,E2 -24535.377} C_VEL
LIN {X 0,Y 155.606,Z 533.676,A -85,B 0,C 180,E1 -24539.11,E2 -24539.11} C_VEL
LIN {X 0,Y 150.434,Z 539.547,A -85,B 0,C 180,E1 -24543.652,E2 -24543.652} C_VEL
LIN {X 0,Y 146.999,Z 543.035,A -85,B 0,C 180,E1 -24547.513,E2 -24547.513} C_VEL
LIN {X 0,Y 145.065,Z 544.812,A -85,B 0,C 180,E1 -24550.176,E2 -24550.176} C_VEL
LIN {X 0,Y 142.343,Z 547.156,A -85,B 0,C 180,E1 -24555.707,E2 -24555.707} C_VEL
LIN {X 0,Y 140.908,Z 547.965,A -85,B 0,C 180,E1 -24561.394,E2 -24561.394} C_VEL
LIN {X 0,Y 140.587,Z 547.176,A -85,B 0,C 180,E1 -24567.134,E2 -24567.134} C_VEL
LIN {X 0,Y 140.69,Z 546.204,A -85,B 0,C 180,E1 -24569.999,E2 -24569.999} C_VEL
LIN {X 0,Y 140.55,Z 544.797,A -85,B 0,C 180,E1 -24572.866,E2 -24572.866} C_VEL
LIN {X 0,Y 140.738,Z 541.843,A -85,B 0,C 180,E1 -24577.171,E2 -24577.171} C_VEL
LIN {X 0,Y 141.384,Z 537.817,A -85,B 0,C 180,E1 -24581.468,E2 -24581.468} C_VEL
LIN {X 0,Y 142.831,Z 531.583,A -85,B 0,C 180,E1 -24586.434,E2 -24586.434} C_VEL
LIN {X 0,Y 144.996,Z 524.79,A -85,B 0,C 180,E1 -24590.572,E2 -24590.572} C_VEL
LIN {X 0,Y 147.636,Z 516.307,A -85,B 0,C 180,E1 -24594.615,E2 -24594.615} C_VEL
LIN {X 0,Y 150.051,Z 508.728,A -85,B 0,C 180,E1 -24597.469,E2 -24597.469} C_VEL
LIN {X 0,Y 152.049,Z 501.324,A -85,B 0,C 180,E1 -24599.793,E2 -24599.793} C_VEL
LIN {X 0,Y 152.637,Z 491.163,A -85,B 0,C 180,E1 -24602.751,E2 -24602.751} C_VEL
LIN {X 0,Y 152.762,Z 481.673,A -85,B 0,C 180,E1 -24605.102,E2 -24605.102} C_VEL
LIN {X 0,Y 152.066,Z 471.097,A -85,B 0,C 180,E1 -24607.435,E2 -24607.435} C_VEL
LIN {X 0,Y 150.577,Z 459.871,A -85,B 0,C 180,E1 -24609.635,E2 -24609.635} C_VEL
LIN {X 0,Y 149.017,Z 453.455,A -85,B 0,C 180,E1 -24610.88,E2 -24610.88} C_VEL
LIN {X 0,Y 145.626,Z 445.665,A -85,B 0,C 180,E1 -24612.649,E2 -24612.649} C_VEL
LIN {X 0,Y 144.149,Z 442.365,A -85,B 0,C 180,E1 -24613.39,E2 -24613.39} C_VEL
LIN {X 0,Y 143.989,Z 441.577,A -85,B 0,C 180,E1 -24613.558,E2 -24613.558} C_VEL
LIN {X 0,Y 143.604,Z 439.995,A -85,B 0,C 180,E1 -24616.468,E2 -24616.468} C_VEL
LIN {X 0,Y 142.753,Z 439.046,A -85,B 0,C 180,E1 -24618.764,E2 -24618.764} C_VEL
LIN {X 0,Y 141.063,Z 438.573,A -85,B 0,C 180,E1 -24621.05,E2 -24621.05} C_VEL
LIN {X 0,Y 136.404,Z 438.516,A -85,B 0,C 180,E1 -24627.398,E2 -24627.398} C_VEL
LIN {X 0,Y 136.054,Z 438.531,A -85,B 0,C 180,E1 -24629.08,E2 -24629.08} C_VEL
LIN {X 0,Y 136.144,Z 438.499,A -85,B 0,C 180,E1 -24632.315,E2 -24632.315} C_VEL
LIN {X 0,Y 136.241,Z 438.51,A -85,B 0,C 180,E1 -24638.832,E2 -24638.832} C_VEL
LIN {X 0,Y 136.262,Z 438.478,A -85,B 0,C 180,E1 -24645.055,E2 -24645.055} C_VEL
LIN {X 0,Y 136.494,Z 438.478,A -85,B 0,C 180,E1 -24648.114,E2 -24648.114} C_VEL
LIN {X 0,Y 136.595,Z 438.467,A -85,B 0,C 180,E1 -24651.12,E2 -24651.12} C_VEL
LIN {X 0,Y 137.131,Z 438.381,A -85,B 0,C 180,E1 -24659.999,E2 -24659.999} C_VEL
LIN {X 0,Y 136.587,Z 438.439,A -85,B 0,C 180,E1 -24668.879,E2 -24668.879} C_VEL
LIN {X 0,Y 136.488,Z 438.437,A -85,B 0,C 180,E1 -24671.954,E2 -24671.954} C_VEL
LIN {X 0,Y 136.238,Z 438.515,A -85,B 0,C 180,E1 -24678.03,E2 -24678.03} C_VEL
LIN {X 0,Y 136.194,Z 438.51,A -85,B 0,C 180,E1 -24681.748,E2 -24681.748} C_VEL
LIN {X 0,Y 136.095,Z 438.521,A -85,B 0,C 180,E1 -24688.615,E2 -24688.615} C_VEL
LIN {X 0,Y 136.08,Z 438.527,A -85,B 0,C 180,E1 -24694.618,E2 -24694.618} C_VEL
LIN {X 0,Y 136.101,Z 438.532,A -85,B 0,C 180,E1 -24699.236,E2 -24699.236} C_VEL
LIN {X 0,Y 136.115,Z 438.528,A -85,B 0,C 180,E1 -24703.711,E2 -24703.711} C_VEL
LIN {X 0,Y 136.115,Z 438.53,A -85,B 0,C 180,E1 -24707.84,E2 -24707.84} C_VEL
LIN {X 0,Y 136.118,Z 438.528,A -85,B 0,C 180,E1 -24711.716,E2 -24711.716} C_VEL
LIN {X 0,Y 136.14,Z 438.527,A -85,B 0,C 180,E1 -24718.272,E2 -24718.272} C_VEL
LIN {X 0,Y 137.1,Z 441.331,A -85,B 0,C 180,E1 -24718.947,E2 -24718.947} C_VEL
LIN {X 0,Y 138.458,Z 443.299,A -85,B 0,C 180,E1 -24719.643,E2 -24719.643} C_VEL
LIN {X 0,Y 143.736,Z 453.04,A -85,B 0,C 180,E1 -24722.625,E2 -24722.625} C_VEL
LIN {X 0,Y 146.34,Z 463.155,A -85,B 0,C 180,E1 -24725.115,E2 -24725.115} C_VEL
LIN {X 0,Y 147.818,Z 474.648,A -85,B 0,C 180,E1 -24728.013,E2 -24728.013} C_VEL
LIN {X 0,Y 148.396,Z 484.01,A -85,B 0,C 180,E1 -24730.64,E2 -24730.64} C_VEL
LIN {X 0,Y 148.266,Z 487.95,A -85,B 0,C 180,E1 -24731.794,E2 -24731.794} C_VEL
LIN {X 0,Y 145.301,Z 497.604,A -85,B 0,C 180,E1 -24734.573,E2 -24734.573} C_VEL
LIN {X 0,Y 142.291,Z 506.663,A -85,B 0,C 180,E1 -24737.883,E2 -24737.883} C_VEL
LIN {X 0,Y 139.188,Z 515.516,A -85,B 0,C 180,E1 -24742.019,E2 -24742.019} C_VEL
LIN {X 0,Y 136.8,Z 522.58,A -85,B 0,C 180,E1 -24746.319,E2 -24746.319} C_VEL
LIN {X 0,Y 134.909,Z 529.037,A -85,B 0,C 180,E1 -24751.493,E2 -24751.493} C_VEL
LIN {X 0,Y 133.856,Z 533.302,A -85,B 0,C 180,E1 -24756.028,E2 -24756.028} C_VEL
LIN {X 0,Y 133.326,Z 535.579,A -85,B 0,C 180,E1 -24759.099,E2 -24759.099} C_VEL
LIN {X 0,Y 133.079,Z 537.356,A -85,B 0,C 180,E1 -24762.196,E2 -24762.196} C_VEL
LIN {X 0,Y 133.114,Z 538.712,A -85,B 0,C 180,E1 -24765.307,E2 -24765.307} C_VEL
LIN {X 0,Y 133.433,Z 539.699,A -85,B 0,C 180,E1 -24768.547,E2 -24768.547} C_VEL
LIN {X 0,Y 133.902,Z 540.188,A -85,B 0,C 180,E1 -24771.556,E2 -24771.556} C_VEL
LIN {X 0,Y 134.718,Z 540.274,A -85,B 0,C 180,E1 -24774.667,E2 -24774.667} C_VEL
LIN {X 0,Y 136.389,Z 539.747,A -85,B 0,C 180,E1 -24778.838,E2 -24778.838} C_VEL
LIN {X 0,Y 139.113,Z 538.028,A -85,B 0,C 180,E1 -24783.76,E2 -24783.76} C_VEL
LIN {X 0,Y 142.142,Z 535.687,A -85,B 0,C 180,E1 -24787.713,E2 -24787.713} C_VEL
LIN {X 0,Y 146.484,Z 531.699,A -85,B 0,C 180,E1 -24792.197,E2 -24792.197} C_VEL
LIN {X 0,Y 151.383,Z 526.629,A -85,B 0,C 180,E1 -24796.183,E2 -24796.183} C_VEL
LIN {X 0,Y 156.604,Z 520.517,A -85,B 0,C 180,E1 -24799.721,E2 -24799.721} C_VEL
LIN {X 0,Y 162.659,Z 512.508,A -85,B 0,C 180,E1 -24803.153,E2 -24803.153} C_VEL
LIN {X 0,Y 164.643,Z 509.564,A -85,B 0,C 180,E1 -24804.197,E2 -24804.197} C_VEL
LIN {X 0,Y 165.699,Z 504.693,A -85,B 0,C 180,E1 -24806.538,E2 -24806.538} C_VEL
LIN {X 0,Y 166.303,Z 498.49,A -85,B 0,C 180,E1 -24809.528,E2 -24809.528} C_VEL
LIN {X 0,Y 166.037,Z 493.234,A -85,B 0,C 180,E1 -24812.251,E2 -24812.251} C_VEL
LIN {X 0,Y 165.07,Z 487.748,A -85,B 0,C 180,E1 -24815.345,E2 -24815.345} C_VEL
LIN {X 0,Y 164.292,Z 484.467,A -85,B 0,C 180,E1 -24817.357,E2 -24817.357} C_VEL
LIN {X 0,Y 163.183,Z 480.663,A -85,B 0,C 180,E1 -24819.846,E2 -24819.846} C_VEL
LIN {X 0,Y 160.734,Z 474.327,A -85,B 0,C 180,E1 -24824.791,E2 -24824.791} C_VEL
LIN {X 0,Y 158.516,Z 469.06,A -85,B 0,C 180,E1 -24829.785,E2 -24829.785} C_VEL
LIN {X 0,Y 156.675,Z 465.317,A -85,B 0,C 180,E1 -24834.853,E2 -24834.853} C_VEL
LIN {X 0,Y 155.931,Z 463.948,A -85,B 0,C 180,E1 -24837.417,E2 -24837.417} C_VEL
LIN {X 0,Y 155.277,Z 463.15,A -85,B 0,C 180,E1 -24840,E2 -24840} C_VEL
LIN {X 0,Y 154.426,Z 462.831,A -85,B 0,C 180,E1 -24845.223,E2 -24845.223} C_VEL
LIN {X 0,Y 154.403,Z 462.938,A -85,B 0,C 180,E1 -24847.849,E2 -24847.849} C_VEL
LIN {X 0,Y 155.567,Z 465.292,A -85,B 0,C 180,E1 -24855.728,E2 -24855.728} C_VEL
LIN {X 0,Y 156.345,Z 466.76,A -85,B 0,C 180,E1 -24858.341,E2 -24858.341} C_VEL
LIN {X 0,Y 156.988,Z 469.278,A -85,B 0,C 180,E1 -24860.987,E2 -24860.987} C_VEL
LIN {X 0,Y 158.174,Z 471.215,A -85,B 0,C 180,E1 -24863.572,E2 -24863.572} C_VEL
LIN {X 0,Y 160.569,Z 477.422,A -85,B 0,C 180,E1 -24868.91,E2 -24868.91} C_VEL
LIN {X 0,Y 162.341,Z 483.099,A -85,B 0,C 180,E1 -24872.797,E2 -24872.797} C_VEL
LIN {X 0,Y 164.129,Z 489.753,A -85,B 0,C 180,E1 -24876.833,E2 -24876.833} C_VEL
LIN {X 0,Y 165.345,Z 496.373,A -85,B 0,C 180,E1 -24880.405,E2 -24880.405} C_VEL
LIN {X 0,Y 165.565,Z 500.423,A -85,B 0,C 180,E1 -24882.338,E2 -24882.338} C_VEL
LIN {X 0,Y 164.61,Z 507.31,A -85,B 0,C 180,E1 -24885.214,E2 -24885.214} C_VEL
LIN {X 0,Y 162.409,Z 515.784,A -85,B 0,C 180,E1 -24888.879,E2 -24888.879} C_VEL
LIN {X 0,Y 161.514,Z 518.355,A -85,B 0,C 180,E1 -24890.073,E2 -24890.073} C_VEL
LIN {X 0,Y 159.81,Z 521.122,A -85,B 0,C 180,E1 -24891.195,E2 -24891.195} C_VEL
LIN {X 0,Y 154.114,Z 528.414,A -85,B 0,C 180,E1 -24894.449,E2 -24894.449} C_VEL
LIN {X 0,Y 148.434,Z 535.142,A -85,B 0,C 180,E1 -24898.613,E2 -24898.613} C_VEL
LIN {X 0,Y 144.101,Z 539.617,A -85,B 0,C 180,E1 -24902.398,E2 -24902.398} C_VEL
LIN {X 0,Y 140.463,Z 543.043,A -85,B 0,C 180,E1 -24906.405,E2 -24906.405} C_VEL
LIN {X 0,Y 136.72,Z 546.09,A -85,B 0,C 180,E1 -24912.035,E2 -24912.035} C_VEL
LIN {X 0,Y 134.493,Z 547.598,A -85,B 0,C 180,E1 -24917.935,E2 -24917.935} C_VEL
LIN {X 0,Y 133.55,Z 547.505,A -85,B 0,C 180,E1 -24923.958,E2 -24923.958} C_VEL
LIN {X 0,Y 133.544,Z 546.146,A -85,B 0,C 180,E1 -24929.277,E2 -24929.277} C_VEL
LIN {X 0,Y 133.468,Z 544.412,A -85,B 0,C 180,E1 -24933.018,E2 -24933.018} C_VEL
LIN {X 0,Y 133.676,Z 541.392,A -85,B 0,C 180,E1 -24937.552,E2 -24937.552} C_VEL
LIN {X 0,Y 134.411,Z 537.29,A -85,B 0,C 180,E1 -24942.072,E2 -24942.072} C_VEL
LIN {X 0,Y 136.006,Z 530.964,A -85,B 0,C 180,E1 -24947.284,E2 -24947.284} C_VEL
LIN {X 0,Y 138.326,Z 524.077,A -85,B 0,C 180,E1 -24951.613,E2 -24951.613} C_VEL
LIN {X 0,Y 140.677,Z 517.019,A -85,B 0,C 180,E1 -24955.127,E2 -24955.127} C_VEL
LIN {X 0,Y 142.75,Z 510.663,A -85,B 0,C 180,E1 -24957.725,E2 -24957.725} C_VEL
LIN {X 0,Y 145.304,Z 502.412,A -85,B 0,C 180,E1 -24960.52,E2 -24960.52} C_VEL
LIN {X 0,Y 146.119,Z 491.282,A -85,B 0,C 180,E1 -24963.949,E2 -24963.949} C_VEL
LIN {X 0,Y 146.3,Z 482.179,A -85,B 0,C 180,E1 -24966.335,E2 -24966.335} C_VEL
LIN {X 0,Y 145.735,Z 471.569,A -85,B 0,C 180,E1 -24968.822,E2 -24968.822} C_VEL
LIN {X 0,Y 144.38,Z 460.891,A -85,B 0,C 180,E1 -24971.079,E2 -24971.079} C_VEL
LIN {X 0,Y 143.019,Z 455.993,A -85,B 0,C 180,E1 -24972.186,E2 -24972.186} C_VEL
LIN {X 0,Y 140.473,Z 449.789,A -85,B 0,C 180,E1 -24973.753,E2 -24973.753} C_VEL
LIN {X 0,Y 138.461,Z 445.543,A -85,B 0,C 180,E1 -24974.864,E2 -24974.864} C_VEL
LIN {X 0,Y 136.893,Z 442.45,A -85,B 0,C 180,E1 -24975.708,E2 -24975.708} C_VEL
LIN {X 0,Y 136.667,Z 441.36,A -85,B 0,C 180,E1 -24975.922,E2 -24975.922} C_VEL
LIN {X 0,Y 136.107,Z 438.535,A -85,B 0,C 180,E1 -24981.71,E2 -24981.71} C_VEL
LIN {X 0,Y 136.053,Z 438.538,A -85,B 0,C 180,E1 -24985.738,E2 -24985.738} C_VEL
LIN {X 0,Y 136.054,Z 438.531,A -85,B 0,C 180,E1 -24989.08,E2 -24989.08} C_VEL
LIN {X 0,Y 135.349,Z 438.605,A -85,B 0,C 180,E1 -24991.554,E2 -24991.554} C_VEL
LIN {X 0,Y 133.782,Z 438.809,A -85,B 0,C 180,E1 -24993.996,E2 -24993.996} C_VEL
LIN {X 0,Y 129.383,Z 439.346,A -85,B 0,C 180,E1 -25000.733,E2 -25000.733} C_VEL
LIN {X 0,Y 129.101,Z 439.365,A -85,B 0,C 180,E1 -25002.51,E2 -25002.51} C_VEL
LIN {X 0,Y 129.414,Z 439.359,A -85,B 0,C 180,E1 -25007.819,E2 -25007.819} C_VEL
LIN {X 0,Y 129.519,Z 439.35,A -85,B 0,C 180,E1 -25010.631,E2 -25010.631} C_VEL
LIN {X 0,Y 130.086,Z 439.257,A -85,B 0,C 180,E1 -25019.999,E2 -25019.999} C_VEL
LIN {X 0,Y 129.513,Z 439.313,A -85,B 0,C 180,E1 -25029.369,E2 -25029.369} C_VEL
LIN {X 0,Y 129.389,Z 439.323,A -85,B 0,C 180,E1 -25032.548,E2 -25032.548} C_VEL
LIN {X 0,Y 129.149,Z 439.397,A -85,B 0,C 180,E1 -25039.056,E2 -25039.056} C_VEL
LIN {X 0,Y 129.105,Z 439.393,A -85,B 0,C 180,E1 -25042.398,E2 -25042.398} C_VEL
LIN {X 0,Y 129.025,Z 439.414,A -85,B 0,C 180,E1 -25045.833,E2 -25045.833} C_VEL
LIN {X 0,Y 129.013,Z 439.403,A -85,B 0,C 180,E1 -25049.358,E2 -25049.358} C_VEL
LIN {X 0,Y 129.025,Z 439.403,A -85,B 0,C 180,E1 -25055.212,E2 -25055.212} C_VEL
LIN {X 0,Y 129.046,Z 439.408,A -85,B 0,C 180,E1 -25060.808,E2 -25060.808} C_VEL
LIN {X 0,Y 129.037,Z 439.412,A -85,B 0,C 180,E1 -25065.075,E2 -25065.075} C_VEL
LIN {X 0,Y 129.048,Z 439.409,A -85,B 0,C 180,E1 -25069.68,E2 -25069.68} C_VEL
LIN {X 0,Y 129.067,Z 439.478,A -85,B 0,C 180,E1 -25075.742,E2 -25075.742} C_VEL
LIN {X 0,Y 130.112,Z 442.34,A -85,B 0,C 180,E1 -25076.498,E2 -25076.498} C_VEL
LIN {X 0,Y 131.656,Z 444.429,A -85,B 0,C 180,E1 -25077.386,E2 -25077.386} C_VEL
LIN {X 0,Y 137.449,Z 455.364,A -85,B 0,C 180,E1 -25081.12,E2 -25081.12} C_VEL
LIN {X 0,Y 138.945,Z 459.151,A -85,B 0,C 180,E1 -25082.275,E2 -25082.275} C_VEL
LIN {X 0,Y 140.667,Z 468.181,A -85,B 0,C 180,E1 -25084.665,E2 -25084.665} C_VEL
LIN {X 0,Y 141.691,Z 479.312,A -85,B 0,C 180,E1 -25087.778,E2 -25087.778} C_VEL
LIN {X 0,Y 141.828,Z 487.532,A -85,B 0,C 180,E1 -25090.305,E2 -25090.305} C_VEL
LIN {X 0,Y 141.337,Z 490.147,A -85,B 0,C 180,E1 -25091.086,E2 -25091.086} C_VEL
LIN {X 0,Y 137.807,Z 500.855,A -85,B 0,C 180,E1 -25094.471,E2 -25094.471} C_VEL
LIN {X 0,Y 134.723,Z 509.378,A -85,B 0,C 180,E1 -25097.957,E2 -25097.957} C_VEL
LIN {X 0,Y 131.641,Z 517.684,A -85,B 0,C 180,E1 -25102.331,E2 -25102.331} C_VEL
LIN {X 0,Y 129.386,Z 524.363,A -85,B 0,C 180,E1 -25106.887,E2 -25106.887} C_VEL
LIN {X 0,Y 127.756,Z 529.697,A -85,B 0,C 180,E1 -25111.577,E2 -25111.577} C_VEL
LIN {X 0,Y 126.67,Z 533.863,A -85,B 0,C 180,E1 -25116.371,E2 -25116.371} C_VEL
LIN {X 0,Y 126.174,Z 536.05,A -85,B 0,C 180,E1 -25119.62,E2 -25119.62} C_VEL
LIN {X 0,Y 125.954,Z 537.773,A -85,B 0,C 180,E1 -25122.897,E2 -25122.897} C_VEL
LIN {X 0,Y 126.376,Z 539.875,A -85,B 0,C 180,E1 -25129.022,E2 -25129.022} C_VEL
LIN {X 0,Y 127.05,Z 540.423,A -85,B 0,C 180,E1 -25132.782,E2 -25132.782} C_VEL
LIN {X 0,Y 128.037,Z 540.462,A -85,B 0,C 180,E1 -25136.048,E2 -25136.048} C_VEL
LIN {X 0,Y 129.643,Z 539.985,A -85,B 0,C 180,E1 -25139.847,E2 -25139.847} C_VEL
LIN {X 0,Y 132.969,Z 538.028,A -85,B 0,C 180,E1 -25145.549,E2 -25145.549} C_VEL
LIN {X 0,Y 135.837,Z 535.984,A -85,B 0,C 180,E1 -25149.098,E2 -25149.098} C_VEL
LIN {X 0,Y 141.053,Z 531.494,A -85,B 0,C 180,E1 -25154.231,E2 -25154.231} C_VEL
LIN {X 0,Y 146.166,Z 526.471,A -85,B 0,C 180,E1 -25158.18,E2 -25158.18} C_VEL
LIN {X 0,Y 151.938,Z 520.08,A -85,B 0,C 180,E1 -25161.845,E2 -25161.845} C_VEL
LIN {X 0,Y 157.022,Z 513.619,A -85,B 0,C 180,E1 -25164.656,E2 -25164.656} C_VEL
LIN {X 0,Y 158.248,Z 511.99,A -85,B 0,C 180,E1 -25165.243,E2 -25165.243} C_VEL
LIN {X 0,Y 159.091,Z 510.412,A -85,B 0,C 180,E1 -25165.922,E2 -25165.922} C_VEL
LIN {X 0,Y 160.269,Z 504.596,A -85,B 0,C 180,E1 -25168.987,E2 -25168.987} C_VEL
LIN {X 0,Y 160.684,Z 499.186,A -85,B 0,C 180,E1 -25171.887,E2 -25171.887} C_VEL
LIN {X 0,Y 160.219,Z 493.355,A -85,B 0,C 180,E1 -25175.373,E2 -25175.373} C_VEL
LIN {X 0,Y 158.959,Z 487.615,A -85,B 0,C 180,E1 -25179.287,E2 -25179.287} C_VEL
LIN {X 0,Y 158.618,Z 485.69,A -85,B 0,C 180,E1 -25180.592,E2 -25180.592} C_VEL
LIN {X 0,Y 156.631,Z 479.61,A -85,B 0,C 180,E1 -25185.713,E2 -25185.713} C_VEL
LIN {X 0,Y 154.811,Z 474.71,A -85,B 0,C 180,E1 -25190.858,E2 -25190.858} C_VEL
LIN {X 0,Y 153.676,Z 471.986,A -85,B 0,C 180,E1 -25194.753,E2 -25194.753} C_VEL
LIN {X 0,Y 153.094,Z 470.549,A -85,B 0,C 180,E1 -25197.369,E2 -25197.369} C_VEL
LIN {X 0,Y 152.514,Z 469.7,A -85,B 0,C 180,E1 -25200,E2 -25200} C_VEL
LIN {X 0,Y 151.708,Z 469.395,A -85,B 0,C 180,E1 -25205.317,E2 -25205.317} C_VEL
LIN {X 0,Y 151.684,Z 469.555,A -85,B 0,C 180,E1 -25207.99,E2 -25207.99} C_VEL
LIN {X 0,Y 152.385,Z 471.395,A -85,B 0,C 180,E1 -25214.418,E2 -25214.418} C_VEL
LIN {X 0,Y 152.78,Z 472.043,A -85,B 0,C 180,E1 -25216.022,E2 -25216.022} C_VEL
LIN {X 0,Y 153.55,Z 474.925,A -85,B 0,C 180,E1 -25219.92,E2 -25219.92} C_VEL
LIN {X 0,Y 154.546,Z 477.015,A -85,B 0,C 180,E1 -25222.74,E2 -25222.74} C_VEL
LIN {X 0,Y 156.341,Z 482.407,A -85,B 0,C 180,E1 -25227.788,E2 -25227.788} C_VEL
LIN {X 0,Y 157.69,Z 487.447,A -85,B 0,C 180,E1 -25231.58,E2 -25231.58} C_VEL
LIN {X 0,Y 158.879,Z 492.742,A -85,B 0,C 180,E1 -25235.104,E2 -25235.104} C_VEL
LIN {X 0,Y 159.853,Z 499.615,A -85,B 0,C 180,E1 -25239.174,E2 -25239.174} C_VEL
LIN {X 0,Y 159.995,Z 503.461,A -85,B 0,C 180,E1 -25241.216,E2 -25241.216} C_VEL
LIN {X 0,Y 158.392,Z 511.309,A -85,B 0,C 180,E1 -25244.771,E2 -25244.771} C_VEL
LIN {X 0,Y 155.886,Z 518.808,A -85,B 0,C 180,E1 -25248.319,E2 -25248.319} C_VEL
LIN {X 0,Y 155.286,Z 520.159,A -85,B 0,C 180,E1 -25248.986,E2 -25248.986} C_VEL
LIN {X 0,Y 149.353,Z 527.577,A -85,B 0,C 180,E1 -25252.286,E2 -25252.286} C_VEL
LIN {X 0,Y 143.879,Z 533.743,A -85,B 0,C 180,E1 -25255.993,E2 -25255.993} C_VEL
LIN {X 0,Y 139.34,Z 538.329,A -85,B 0,C 180,E1 -25259.71,E2 -25259.71} C_VEL
LIN {X 0,Y 135.192,Z 542.013,A -85,B 0,C 180,E1 -25263.776,E2 -25263.776} C_VEL
LIN {X 0,Y 131.784,Z 544.713,A -85,B 0,C 180,E1 -25268.08,E2 -25268.08} C_VEL
LIN {X 0,Y 128.587,Z 546.917,A -85,B 0,C 180,E1 -25274.14,E2 -25274.14} C_VEL
LIN {X 0,Y 126.861,Z 547.521,A -85,B 0,C 180,E1 -25280.433,E2 -25280.433} C_VEL
LIN {X 0,Y 126.439,Z 546.601,A -85,B 0,C 180,E1 -25286.813,E2 -25286.813} C_VEL
LIN {X 0,Y 126.505,Z 545.545,A -85,B 0,C 180,E1 -25289.999,E2 -25289.999} C_VEL
LIN {X 0,Y 126.38,Z 544.017,A -85,B 0,C 180,E1 -25293.187,E2 -25293.187} C_VEL
LIN {X 0,Y 126.637,Z 540.922,A -85,B 0,C 180,E1 -25297.974,E2 -25297.974} C_VEL
LIN {X 0,Y 127.434,Z 536.738,A -85,B 0,C 180,E1 -25302.743,E2 -25302.743} C_VEL
LIN {X 0,Y 129.215,Z 530.326,A -85,B 0,C 180,E1 -25308.224,E2 -25308.224} C_VEL
LIN {X 0,Y 131.693,Z 523.334,A -85,B 0,C 180,E1 -25312.761,E2 -25312.761} C_VEL
LIN {X 0,Y 134.05,Z 516.501,A -85,B 0,C 180,E1 -25316.274,E2 -25316.274} C_VEL
LIN {X 0,Y 137.183,Z 507.657,A -85,B 0,C 180,E1 -25319.881,E2 -25319.881} C_VEL
LIN {X 0,Y 138.716,Z 502.34,A -85,B 0,C 180,E1 -25321.71,E2 -25321.71} C_VEL
LIN {X 0,Y 139.59,Z 492.129,A -85,B 0,C 180,E1 -25325.039,E2 -25325.039} C_VEL
LIN {X 0,Y 139.908,Z 482.423,A -85,B 0,C 180,E1 -25327.751,E2 -25327.751} C_VEL
LIN {X 0,Y 139.38,Z 471.126,A -85,B 0,C 180,E1 -25330.565,E2 -25330.565} C_VEL
LIN {X 0,Y 138.33,Z 462.425,A -85,B 0,C 180,E1 -25332.547,E2 -25332.547} C_VEL
LIN {X 0,Y 136.299,Z 456.245,A -85,B 0,C 180,E1 -25334.197,E2 -25334.197} C_VEL
LIN {X 0,Y 133.287,Z 449.469,A -85,B 0,C 180,E1 -25336.183,E2 -25336.183} C_VEL
LIN {X 0,Y 131.339,Z 445.572,A -85,B 0,C 180,E1 -25337.371,E2 -25337.371} C_VEL
LIN {X 0,Y 129.65,Z 442.357,A -85,B 0,C 180,E1 -25338.391,E2 -25338.391} C_VEL
LIN {X 0,Y 129.327,Z 441.054,A -85,B 0,C 180,E1 -25338.783,E2 -25338.783} C_VEL
LIN {X 0,Y 128.992,Z 439.421,A -85,B 0,C 180,E1 -25342.689,E2 -25342.689} C_VEL
LIN {X 0,Y 128.974,Z 439.42,A -85,B 0,C 180,E1 -25346.98,E2 -25346.98} C_VEL
LIN {X 0,Y 129.014,Z 439.393,A -85,B 0,C 180,E1 -25350.641,E2 -25350.641} C_VEL
LIN {X 0,Y 129.027,Z 439.393,A -85,B 0,C 180,E1 -25354.166,E2 -25354.166} C_VEL
LIN {X 0,Y 129.105,Z 439.402,A -85,B 0,C 180,E1 -25357.727,E2 -25357.727} C_VEL
LIN {X 0,Y 129.101,Z 439.365,A -85,B 0,C 180,E1 -25362.51,E2 -25362.51} C_VEL
LIN {X 0,Y 128.465,Z 439.451,A -85,B 0,C 180,E1 -25365.118,E2 -25365.118} C_VEL
LIN {X 0,Y 126.927,Z 439.667,A -85,B 0,C 180,E1 -25367.695,E2 -25367.695} C_VEL
LIN {X 0,Y 123.411,Z 440.094,A -85,B 0,C 180,E1 -25372.979,E2 -25372.979} C_VEL
LIN {X 0,Y 122.587,Z 440.169,A -85,B 0,C 180,E1 -25375.761,E2 -25375.761} C_VEL
LIN {X 0,Y 122.601,Z 440.165,A -85,B 0,C 180,E1 -25376.699,E2 -25376.699} C_VEL
LIN {X 0,Y 123.04,Z 440.132,A -85,B 0,C 180,E1 -25379.999,E2 -25379.999} C_VEL
LIN {X 0,Y 122.414,Z 440.217,A -85,B 0,C 180,E1 -25387.17,E2 -25387.17} C_VEL
LIN {X 0,Y 122.36,Z 440.196,A -85,B 0,C 180,E1 -25392.473,E2 -25392.473} C_VEL
LIN {X 0,Y 122.041,Z 440.278,A -85,B 0,C 180,E1 -25400.213,E2 -25400.213} C_VEL
LIN {X 0,Y 121.979,Z 440.285,A -85,B 0,C 180,E1 -25403.785,E2 -25403.785} C_VEL
LIN {X 0,Y 121.926,Z 440.288,A -85,B 0,C 180,E1 -25410.164,E2 -25410.164} C_VEL
LIN {X 0,Y 121.946,Z 440.284,A -85,B 0,C 180,E1 -25416.214,E2 -25416.214} C_VEL
LIN {X 0,Y 121.966,Z 440.291,A -85,B 0,C 180,E1 -25421.491,E2 -25421.491} C_VEL
LIN {X 0,Y 121.967,Z 440.291,A -85,B 0,C 180,E1 -25428.511,E2 -25428.511} C_VEL
LIN {X 0,Y 121.955,Z 440.307,A -85,B 0,C 180,E1 -25432.727,E2 -25432.727} C_VEL
LIN {X 0,Y 122.997,Z 443.165,A -85,B 0,C 180,E1 -25433.596,E2 -25433.596} C_VEL
LIN {X 0,Y 124.789,Z 445.521,A -85,B 0,C 180,E1 -25434.757,E2 -25434.757} C_VEL
LIN {X 0,Y 126.797,Z 448.843,A -85,B 0,C 180,E1 -25436.135,E2 -25436.135} C_VEL
LIN {X 0,Y 132.414,Z 460.034,A -85,B 0,C 180,E1 -25440.358,E2 -25440.358} C_VEL
LIN {X 0,Y 133.313,Z 462.699,A -85,B 0,C 180,E1 -25441.227,E2 -25441.227} C_VEL
LIN {X 0,Y 134.619,Z 470.786,A -85,B 0,C 180,E1 -25443.571,E2 -25443.571} C_VEL
LIN {X 0,Y 135.348,Z 481.051,A -85,B 0,C 180,E1 -25446.677,E2 -25446.677} C_VEL
LIN {X 0,Y 135.263,Z 489.674,A -85,B 0,C 180,E1 -25449.531,E2 -25449.531} C_VEL
LIN {X 0,Y 131.651,Z 500.194,A -85,B 0,C 180,E1 -25452.927,E2 -25452.927} C_VEL
LIN {X 0,Y 128.358,Z 508.9,A -85,B 0,C 180,E1 -25456.545,E2 -25456.545} C_VEL
LIN {X 0,Y 125.049,Z 517.339,A -85,B 0,C 180,E1 -25461.11,E2 -25461.11} C_VEL
LIN {X 0,Y 122.579,Z 524.119,A -85,B 0,C 180,E1 -25465.891,E2 -25465.891} C_VEL
LIN {X 0,Y 120.6,Z 530.347,A -85,B 0,C 180,E1 -25471.67,E2 -25471.67} C_VEL
LIN {X 0,Y 119.475,Z 534.413,A -85,B 0,C 180,E1 -25476.757,E2 -25476.757} C_VEL
LIN {X 0,Y 119.015,Z 536.514,A -85,B 0,C 180,E1 -25480.205,E2 -25480.205} C_VEL
LIN {X 0,Y 118.848,Z 538.191,A -85,B 0,C 180,E1 -25483.683,E2 -25483.683} C_VEL
LIN {X 0,Y 119.358,Z 540.06,A -85,B 0,C 180,E1 -25489.593,E2 -25489.593} C_VEL
LIN {X 0,Y 120.254,Z 540.658,A -85,B 0,C 180,E1 -25494.148,E2 -25494.148} C_VEL
LIN {X 0,Y 121.417,Z 540.651,A -85,B 0,C 180,E1 -25497.585,E2 -25497.585} C_VEL
LIN {X 0,Y 122.939,Z 540.224,A -85,B 0,C 180,E1 -25500.964,E2 -25500.964} C_VEL
LIN {X 0,Y 124.764,Z 539.334,A -85,B 0,C 180,E1 -25504.285,E2 -25504.285} C_VEL
LIN {X 0,Y 126.994,Z 538.028,A -85,B 0,C 180,E1 -25507.499,E2 -25507.499} C_VEL
LIN {X 0,Y 130.878,Z 535.319,A -85,B 0,C 180,E1 -25511.955,E2 -25511.955} C_VEL
LIN {X 0,Y 135.817,Z 531.289,A -85,B 0,C 180,E1 -25516.422,E2 -25516.422} C_VEL
LIN {X 0,Y 141.306,Z 526.151,A -85,B 0,C 180,E1 -25520.435,E2 -25520.435} C_VEL
LIN {X 0,Y 147.45,Z 519.603,A -85,B 0,C 180,E1 -25524.123,E2 -25524.123} C_VEL
LIN {X 0,Y 152.933,Z 512.856,A -85,B 0,C 180,E1 -25526.999,E2 -25526.999} C_VEL
LIN {X 0,Y 154.411,Z 507.579,A -85,B 0,C 180,E1 -25529.957,E2 -25529.957} C_VEL
LIN {X 0,Y 154.987,Z 504.027,A -85,B 0,C 180,E1 -25531.994,E2 -25531.994} C_VEL
LIN {X 0,Y 155.028,Z 499.236,A -85,B 0,C 180,E1 -25535.048,E2 -25535.048} C_VEL
LIN {X 0,Y 154.473,Z 494.125,A -85,B 0,C 180,E1 -25538.656,E2 -25538.656} C_VEL
LIN {X 0,Y 153.876,Z 490.563,A -85,B 0,C 180,E1 -25541.355,E2 -25541.355} C_VEL
LIN {X 0,Y 152.331,Z 484.767,A -85,B 0,C 180,E1 -25546.663,E2 -25546.663} C_VEL
LIN {X 0,Y 150.915,Z 480.216,A -85,B 0,C 180,E1 -25551.97,E2 -25551.97} C_VEL
LIN {X 0,Y 149.868,Z 476.97,A -85,B 0,C 180,E1 -25557.313,E2 -25557.313} C_VEL
LIN {X 0,Y 149.402,Z 476.085,A -85,B 0,C 180,E1 -25560,E2 -25560} C_VEL
LIN {X 0,Y 148.639,Z 475.802,A -85,B 0,C 180,E1 -25565.427,E2 -25565.427} C_VEL
LIN {X 0,Y 148.61,Z 476.017,A -85,B 0,C 180,E1 -25568.157,E2 -25568.157} C_VEL
LIN {X 0,Y 149.063,Z 477.523,A -85,B 0,C 180,E1 -25573.636,E2 -25573.636} C_VEL
LIN {X 0,Y 149.545,Z 478.71,A -85,B 0,C 180,E1 -25576.379,E2 -25576.379} C_VEL
LIN {X 0,Y 151.066,Z 483.835,A -85,B 0,C 180,E1 -25583.294,E2 -25583.294} C_VEL
LIN {X 0,Y 152.189,Z 488.281,A -85,B 0,C 180,E1 -25587.504,E2 -25587.504} C_VEL
LIN {X 0,Y 153.172,Z 493.121,A -85,B 0,C 180,E1 -25591.349,E2 -25591.349} C_VEL
LIN {X 0,Y 154.053,Z 499.111,A -85,B 0,C 180,E1 -25595.536,E2 -25595.536} C_VEL
LIN {X 0,Y 154.442,Z 505.128,A -85,B 0,C 180,E1 -25599.323,E2 -25599.323} C_VEL
LIN {X 0,Y 153.758,Z 509.257,A -85,B 0,C 180,E1 -25601.457,E2 -25601.457} C_VEL
LIN {X 0,Y 151.869,Z 515.398,A -85,B 0,C 180,E1 -25604.446,E2 -25604.446} C_VEL
LIN {X 0,Y 149.79,Z 520.55,A -85,B 0,C 180,E1 -25607.131,E2 -25607.131} C_VEL
LIN {X 0,Y 149.012,Z 521.875,A -85,B 0,C 180,E1 -25607.772,E2 -25607.772} C_VEL
LIN {X 0,Y 142.82,Z 528.95,A -85,B 0,C 180,E1 -25611.141,E2 -25611.141} C_VEL
LIN {X 0,Y 136.662,Z 535.262,A -85,B 0,C 180,E1 -25615.369,E2 -25615.369} C_VEL
LIN {X 0,Y 131.685,Z 539.739,A -85,B 0,C 180,E1 -25619.535,E2 -25619.535} C_VEL
LIN {X 0,Y 127.561,Z 543.017,A -85,B 0,C 180,E1 -25623.848,E2 -25623.848} C_VEL
LIN {X 0,Y 123.23,Z 545.921,A -85,B 0,C 180,E1 -25629.989,E2 -25629.989} C_VEL
LIN {X 0,Y 121.741,Z 546.783,A -85,B 0,C 180,E1 -25633.223,E2 -25633.223} C_VEL
LIN {X 0,Y 119.846,Z 547.298,A -85,B 0,C 180,E1 -25639.867,E2 -25639.867} C_VEL
LIN {X 0,Y 119.353,Z 546.309,A -85,B 0,C 180,E1 -25646.624,E2 -25646.624} C_VEL
LIN {X 0,Y 119.418,Z 545.186,A -85,B 0,C 180,E1 -25649.999,E2 -25649.999} C_VEL
LIN {X 0,Y 119.287,Z 543.62,A -85,B 0,C 180,E1 -25653.377,E2 -25653.377} C_VEL
LIN {X 0,Y 119.599,Z 540.45,A -85,B 0,C 180,E1 -25658.447,E2 -25658.447} C_VEL
LIN {X 0,Y 120.486,Z 536.185,A -85,B 0,C 180,E1 -25663.492,E2 -25663.492} C_VEL
LIN {X 0,Y 122.466,Z 529.687,A -85,B 0,C 180,E1 -25669.266,E2 -25669.266} C_VEL
LIN {X 0,Y 125.085,Z 522.549,A -85,B 0,C 180,E1 -25674.037,E2 -25674.037} C_VEL
LIN {X 0,Y 127.525,Z 515.868,A -85,B 0,C 180,E1 -25677.592,E2 -25677.592} C_VEL
LIN {X 0,Y 131.128,Z 506.414,A -85,B 0,C 180,E1 -25681.503,E2 -25681.503} C_VEL
LIN {X 0,Y 132.032,Z 503.389,A -85,B 0,C 180,E1 -25682.611,E2 -25682.611} C_VEL
LIN {X 0,Y 133.085,Z 493.413,A -85,B 0,C 180,E1 -25686.097,E2 -25686.097} C_VEL
LIN {X 0,Y 133.624,Z 483.251,A -85,B 0,C 180,E1 -25689.133,E2 -25689.133} C_VEL
LIN {X 0,Y 133.163,Z 471.158,A -85,B 0,C 180,E1 -25692.363,E2 -25692.363} C_VEL
LIN {X 0,Y 132.289,Z 463.985,A -85,B 0,C 180,E1 -25694.173,E2 -25694.173} C_VEL
LIN {X 0,Y 129.004,Z 455.012,A -85,B 0,C 180,E1 -25696.945,E2 -25696.945} C_VEL
LIN {X 0,Y 124.874,Z 446.429,A -85,B 0,C 180,E1 -25699.891,E2 -25699.891} C_VEL
LIN {X 0,Y 122.645,Z 442.658,A -85,B 0,C 180,E1 -25701.359,E2 -25701.359} C_VEL
LIN {X 0,Y 122.071,Z 440.808,A -85,B 0,C 180,E1 -25701.905,E2 -25701.905} C_VEL
LIN {X 0,Y 121.913,Z 440.301,A -85,B 0,C 180,E1 -25703.807,E2 -25703.807} C_VEL
LIN {X 0,Y 121.924,Z 440.283,A -85,B 0,C 180,E1 -25709.838,E2 -25709.838} C_VEL
LIN {X 0,Y 121.981,Z 440.287,A -85,B 0,C 180,E1 -25716.214,E2 -25716.214} C_VEL
LIN {X 0,Y 122.046,Z 440.242,A -85,B 0,C 180,E1 -25722.597,E2 -25722.597} C_VEL
LIN {X 0,Y 122.361,Z 440.233,A -85,B 0,C 180,E1 -25727.525,E2 -25727.525} C_VEL
LIN {X 0,Y 122.447,Z 440.233,A -85,B 0,C 180,E1 -25730.084,E2 -25730.084} C_VEL
LIN {X 0,Y 122.601,Z 440.165,A -85,B 0,C 180,E1 -25736.699,E2 -25736.699} C_VEL
LIN {X 0,Y 122.432,Z 440.194,A -85,B 0,C 180,E1 -25738.528,E2 -25738.528} C_VEL
LIN {X 0,Y 121.16,Z 440.38,A -85,B 0,C 180,E1 -25741.24,E2 -25741.24} C_VEL
LIN {X 0,Y 115.696,Z 441.03,A -85,B 0,C 180,E1 -25749.632,E2 -25749.632} C_VEL
LIN {X 0,Y 115.299,Z 441.071,A -85,B 0,C 180,E1 -25751.635,E2 -25751.635} C_VEL
LIN {X 0,Y 115.008,Z 441.158,A -85,B 0,C 180,E1 -25757.79,E2 -25757.79} C_VEL
LIN {X 0,Y 114.944,Z 441.16,A -85,B 0,C 180,E1 -25763.492,E2 -25763.492} C_VEL
LIN {X 0,Y 114.861,Z 441.174,A -85,B 0,C 180,E1 -25771.064,E2 -25771.064} C_VEL
LIN {X 0,Y 114.879,Z 441.171,A -85,B 0,C 180,E1 -25777.717,E2 -25777.717} C_VEL
LIN {X 0,Y 114.884,Z 441.173,A -85,B 0,C 180,E1 -25782.771,E2 -25782.771} C_VEL
LIN {X 0,Y 114.928,Z 441.213,A -85,B 0,C 180,E1 -25789.216,E2 -25789.216} C_VEL
LIN {X 0,Y 115.783,Z 443.81,A -85,B 0,C 180,E1 -25790.103,E2 -25790.103} C_VEL
LIN {X 0,Y 117.876,Z 446.463,A -85,B 0,C 180,E1 -25791.671,E2 -25791.671} C_VEL
LIN {X 0,Y 119.735,Z 449.689,A -85,B 0,C 180,E1 -25793.174,E2 -25793.174} C_VEL
LIN {X 0,Y 124.072,Z 457.692,A -85,B 0,C 180,E1 -25796.723,E2 -25796.723} C_VEL
LIN {X 0,Y 127.388,Z 464.866,A -85,B 0,C 180,E1 -25799.684,E2 -25799.684} C_VEL
LIN {X 0,Y 128.68,Z 474.345,A -85,B 0,C 180,E1 -25802.678,E2 -25802.678} C_VEL
LIN {X 0,Y 129.082,Z 484.05,A -85,B 0,C 180,E1 -25805.9,E2 -25805.9} C_VEL
LIN {X 0,Y 128.942,Z 489.643,A -85,B 0,C 180,E1 -25807.907,E2 -25807.907} C_VEL
LIN {X 0,Y 127.439,Z 494.574,A -85,B 0,C 180,E1 -25809.492,E2 -25809.492} C_VEL
LIN {X 0,Y 123.422,Z 505.073,A -85,B 0,C 180,E1 -25813.459,E2 -25813.459} C_VEL
LIN {X 0,Y 119.604,Z 514.32,A -85,B 0,C 180,E1 -25818.133,E2 -25818.133} C_VEL
LIN {X 0,Y 116.586,Z 521.75,A -85,B 0,C 180,E1 -25823.076,E2 -25823.076} C_VEL
LIN {X 0,Y 114.456,Z 527.701,A -85,B 0,C 180,E1 -25828.241,E2 -25828.241} C_VEL
LIN {X 0,Y 113.001,Z 532.41,A -85,B 0,C 180,E1 -25833.566,E2 -25833.566} C_VEL
LIN {X 0,Y 112.052,Z 536.022,A -85,B 0,C 180,E1 -25839.022,E2 -25839.022} C_VEL
LIN {X 0,Y 111.775,Z 538.609,A -85,B 0,C 180,E1 -25844.567,E2 -25844.567} C_VEL
LIN {X 0,Y 112.366,Z 540.249,A -85,B 0,C 180,E1 -25850.253,E2 -25850.253} C_VEL
LIN {X 0,Y 113.542,Z 540.894,A -85,B 0,C 180,E1 -25855.676,E2 -25855.676} C_VEL
LIN {X 0,Y 116.298,Z 540.458,A -85,B 0,C 180,E1 -25862.218,E2 -25862.218} C_VEL
LIN {X 0,Y 118.67,Z 539.383,A -85,B 0,C 180,E1 -25866.315,E2 -25866.315} C_VEL
LIN {X 0,Y 123.505,Z 536.565,A -85,B 0,C 180,E1 -25872.29,E2 -25872.29} C_VEL
LIN {X 0,Y 128.982,Z 532.546,A -85,B 0,C 180,E1 -25877.357,E2 -25877.357} C_VEL
LIN {X 0,Y 134.651,Z 527.696,A -85,B 0,C 180,E1 -25881.528,E2 -25881.528} C_VEL
LIN {X 0,Y 140.99,Z 521.499,A -85,B 0,C 180,E1 -25885.333,E2 -25885.333} C_VEL
LIN {X 0,Y 146.342,Z 515.505,A -85,B 0,C 180,E1 -25888.112,E2 -25888.112} C_VEL
LIN {X 0,Y 147.555,Z 513.67,A -85,B 0,C 180,E1 -25889.018,E2 -25889.018} C_VEL
LIN {X 0,Y 148.887,Z 509.122,A -85,B 0,C 180,E1 -25891.834,E2 -25891.834} C_VEL
LIN {X 0,Y 149.498,Z 504.419,A -85,B 0,C 180,E1 -25894.97,E2 -25894.97} C_VEL
LIN {X 0,Y 149.434,Z 500.482,A -85,B 0,C 180,E1 -25897.899,E2 -25897.899} C_VEL
LIN {X 0,Y 148.963,Z 495.271,A -85,B 0,C 180,E1 -25902.142,E2 -25902.142} C_VEL
LIN {X 0,Y 148.1,Z 491.054,A -85,B 0,C 180,E1 -25906.275,E2 -25906.275} C_VEL
LIN {X 0,Y 147.07,Z 486.452,A -85,B 0,C 180,E1 -25911.758,E2 -25911.758} C_VEL
LIN {X 0,Y 146.261,Z 483.209,A -85,B 0,C 180,E1 -25917.246,E2 -25917.246} C_VEL
LIN {X 0,Y 145.9,Z 482.289,A -85,B 0,C 180,E1 -25920,E2 -25920} C_VEL
LIN {X 0,Y 145.214,Z 482.035,A -85,B 0,C 180,E1 -25925.555,E2 -25925.555} C_VEL
LIN {X 0,Y 145.188,Z 482.283,A -85,B 0,C 180,E1 -25928.35,E2 -25928.35} C_VEL
LIN {X 0,Y 145.543,Z 483.867,A -85,B 0,C 180,E1 -25933.972,E2 -25933.972} C_VEL
LIN {X 0,Y 145.887,Z 485.258,A -85,B 0,C 180,E1 -25936.801,E2 -25936.801} C_VEL
LIN {X 0,Y 146.879,Z 489.218,A -85,B 0,C 180,E1 -25942.507,E2 -25942.507} C_VEL
LIN {X 0,Y 147.676,Z 493.507,A -85,B 0,C 180,E1 -25946.88,E2 -25946.88} C_VEL
LIN {X 0,Y 148.415,Z 499.016,A -85,B 0,C 180,E1 -25951.531,E2 -25951.531} C_VEL
LIN {X 0,Y 148.81,Z 504.473,A -85,B 0,C 180,E1 -25955.564,E2 -25955.564} C_VEL
LIN {X 0,Y 148.713,Z 509.269,A -85,B 0,C 180,E1 -25958.769,E2 -25958.769} C_VEL
LIN {X 0,Y 147.121,Z 514.633,A -85,B 0,C 180,E1 -25961.654,E2 -25961.654} C_VEL
LIN {X 0,Y 144.385,Z 520.948,A -85,B 0,C 180,E1 -25965.107,E2 -25965.107} C_VEL
LIN {X 0,Y 143.72,Z 522.254,A -85,B 0,C 180,E1 -25965.827,E2 -25965.827} C_VEL
LIN {X 0,Y 137.356,Z 529.182,A -85,B 0,C 180,E1 -25969.28,E2 -25969.28} C_VEL
LIN {X 0,Y 130.535,Z 535.717,A -85,B 0,C 180,E1 -25973.863,E2 -25973.863} C_VEL
LIN {X 0,Y 125.619,Z 539.801,A -85,B 0,C 180,E1 -25977.893,E2 -25977.893} C_VEL
LIN {X 0,Y 121.198,Z 543.004,A -85,B 0,C 180,E1 -25982.361,E2 -25982.361} C_VEL
LIN {X 0,Y 116.556,Z 545.834,A -85,B 0,C 180,E1 -25988.79,E2 -25988.79} C_VEL
LIN {X 0,Y 113.696,Z 547.04,A -85,B 0,C 180,E1 -25995.684,E2 -25995.684} C_VEL
LIN {X 0,Y 112.352,Z 546.736,A -85,B 0,C 180,E1 -26002.813,E2 -26002.813} C_VEL
LIN {X 0,Y 112.262,Z 545.999,A -85,B 0,C 180,E1 -26006.41,E2 -26006.41} C_VEL
LIN {X 0,Y 112.333,Z 544.827,A -85,B 0,C 180,E1 -26009.999,E2 -26009.999} C_VEL
LIN {X 0,Y 112.229,Z 542.264,A -85,B 0,C 180,E1 -26015.389,E2 -26015.389} C_VEL
LIN {X 0,Y 112.809,Z 538.667,A -85,B 0,C 180,E1 -26020.771,E2 -26020.771} C_VEL
LIN {X 0,Y 114.023,Z 533.921,A -85,B 0,C 180,E1 -26026.102,E2 -26026.102} C_VEL
LIN {X 0,Y 116.654,Z 526.779,A -85,B 0,C 180,E1 -26032.118,E2 -26032.118} C_VEL
LIN {X 0,Y 119.769,Z 518.987,A -85,B 0,C 180,E1 -26037.049,E2 -26037.049} C_VEL
LIN {X 0,Y 122.471,Z 511.898,A -85,B 0,C 180,E1 -26040.595,E2 -26040.595} C_VEL
LIN {X 0,Y 125.355,Z 504.358,A -85,B 0,C 180,E1 -26043.616,E2 -26043.616} C_VEL
LIN {X 0,Y 126.74,Z 493.706,A -85,B 0,C 180,E1 -26047.586,E2 -26047.586} C_VEL
LIN {X 0,Y 127.378,Z 484.032,A -85,B 0,C 180,E1 -26050.679,E2 -26050.679} C_VEL
LIN {X 0,Y 127.17,Z 472.118,A -85,B 0,C 180,E1 -26054.073,E2 -26054.073} C_VEL
LIN {X 0,Y 126.492,Z 466.619,A -85,B 0,C 180,E1 -26055.622,E2 -26055.622} C_VEL
LIN {X 0,Y 123.925,Z 459.138,A -85,B 0,C 180,E1 -26058.212,E2 -26058.212} C_VEL
LIN {X 0,Y 119.711,Z 450.151,A -85,B 0,C 180,E1 -26061.676,E2 -26061.676} C_VEL
LIN {X 0,Y 117.521,Z 445.838,A -85,B 0,C 180,E1 -26063.43,E2 -26063.43} C_VEL
LIN {X 0,Y 115.655,Z 443.603,A -85,B 0,C 180,E1 -26064.739,E2 -26064.739} C_VEL
LIN {X 0,Y 114.845,Z 441.181,A -85,B 0,C 180,E1 -26065.656,E2 -26065.656} C_VEL
LIN {X 0,Y 114.855,Z 441.154,A -85,B 0,C 180,E1 -26070.69,E2 -26070.69} C_VEL
LIN {X 0,Y 114.945,Z 441.164,A -85,B 0,C 180,E1 -26076.506,E2 -26076.506} C_VEL
LIN {X 0,Y 114.997,Z 441.12,A -85,B 0,C 180,E1 -26082.207,E2 -26082.207} C_VEL
LIN {X 0,Y 115.282,Z 441.112,A -85,B 0,C 180,E1 -26087.26,E2 -26087.26} C_VEL
LIN {X 0,Y 115.389,Z 441.091,A -85,B 0,C 180,E1 -26093.003,E2 -26093.003} C_VEL
LIN {X 0,Y 115.992,Z 441.008,A -85,B 0,C 180,E1 -26099.999,E2 -26099.999} C_VEL
LIN {X 0,Y 115.381,Z 441.096,A -85,B 0,C 180,E1 -26107.06,E2 -26107.06} C_VEL
LIN {X 0,Y 115.299,Z 441.071,A -85,B 0,C 180,E1 -26111.635,E2 -26111.635} C_VEL
LIN {X 0,Y 114.541,Z 441.19,A -85,B 0,C 180,E1 -26114.545,E2 -26114.545} C_VEL
LIN {X 0,Y 112.89,Z 441.421,A -85,B 0,C 180,E1 -26117.416,E2 -26117.416} C_VEL
LIN {X 0,Y 108.127,Z 442.018,A -85,B 0,C 180,E1 -26125.402,E2 -26125.402} C_VEL
LIN {X 0,Y 107.73,Z 442.057,A -85,B 0,C 180,E1 -26127.534,E2 -26127.534} C_VEL
LIN {X 0,Y 107.793,Z 442.058,A -85,B 0,C 180,E1 -26132.053,E2 -26132.053} C_VEL
LIN {X 0,Y 107.783,Z 442.059,A -85,B 0,C 180,E1 -26138.516,E2 -26138.516} C_VEL
LIN {X 0,Y 107.776,Z 442.132,A -85,B 0,C 180,E1 -26144.839,E2 -26144.839} C_VEL
LIN {X 0,Y 108.653,Z 444.704,A -85,B 0,C 180,E1 -26145.944,E2 -26145.944} C_VEL
LIN {X 0,Y 111.032,Z 447.4,A -85,B 0,C 180,E1 -26148.018,E2 -26148.018} C_VEL
LIN {X 0,Y 112.65,Z 450.414,A -85,B 0,C 180,E1 -26149.623,E2 -26149.623} C_VEL
LIN {X 0,Y 114.057,Z 452.647,A -85,B 0,C 180,E1 -26150.896,E2 -26150.896} C_VEL
LIN {X 0,Y 117.907,Z 459.687,A -85,B 0,C 180,E1 -26154.495,E2 -26154.495} C_VEL
LIN {X 0,Y 121.41,Z 467.535,A -85,B 0,C 180,E1 -26158.099,E2 -26158.099} C_VEL
LIN {X 0,Y 122.101,Z 470.47,A -85,B 0,C 180,E1 -26159.215,E2 -26159.215} C_VEL
LIN {X 0,Y 122.736,Z 478.993,A -85,B 0,C 180,E1 -26162.143,E2 -26162.143} C_VEL
LIN {X 0,Y 122.685,Z 489.159,A -85,B 0,C 180,E1 -26165.912,E2 -26165.912} C_VEL
LIN {X 0,Y 122.236,Z 492.174,A -85,B 0,C 180,E1 -26167.032,E2 -26167.032} C_VEL
LIN {X 0,Y 118.874,Z 500.829,A -85,B 0,C 180,E1 -26170.127,E2 -26170.127} C_VEL
LIN {X 0,Y 115.204,Z 509.491,A -85,B 0,C 180,E1 -26174.068,E2 -26174.068} C_VEL
LIN {X 0,Y 111.498,Z 517.89,A -85,B 0,C 180,E1 -26179.101,E2 -26179.101} C_VEL
LIN {X 0,Y 108.703,Z 524.646,A -85,B 0,C 180,E1 -26184.436,E2 -26184.436} C_VEL
LIN {X 0,Y 106.72,Z 530.045,A -85,B 0,C 180,E1 -26190.001,E2 -26190.001} C_VEL
LIN {X 0,Y 105.41,Z 534.273,A -85,B 0,C 180,E1 -26195.738,E2 -26195.738} C_VEL
LIN {X 0,Y 104.71,Z 537.444,A -85,B 0,C 180,E1 -26201.617,E2 -26201.617} C_VEL
LIN {X 0,Y 104.712,Z 539.019,A -85,B 0,C 180,E1 -26205.574,E2 -26205.574} C_VEL
LIN {X 0,Y 105.364,Z 540.43,A -85,B 0,C 180,E1 -26210.962,E2 -26210.962} C_VEL
LIN {X 0,Y 106.912,Z 541.13,A -85,B 0,C 180,E1 -26217.397,E2 -26217.397} C_VEL
LIN {X 0,Y 109.669,Z 540.696,A -85,B 0,C 180,E1 -26223.584,E2 -26223.584} C_VEL
LIN {X 0,Y 112.766,Z 539.431,A -85,B 0,C 180,E1 -26228.553,E2 -26228.553} C_VEL
LIN {X 0,Y 117.47,Z 536.862,A -85,B 0,C 180,E1 -26234.116,E2 -26234.116} C_VEL
LIN {X 0,Y 122.179,Z 533.728,A -85,B 0,C 180,E1 -26238.399,E2 -26238.399} C_VEL
LIN {X 0,Y 128.428,Z 528.883,A -85,B 0,C 180,E1 -26242.991,E2 -26242.991} C_VEL
LIN {X 0,Y 135.746,Z 522.221,A -85,B 0,C 180,E1 -26247.278,E2 -26247.278} C_VEL
LIN {X 0,Y 141.361,Z 516.212,A -85,B 0,C 180,E1 -26250.188,E2 -26250.188} C_VEL
LIN {X 0,Y 142.794,Z 512.873,A -85,B 0,C 180,E1 -26252.364,E2 -26252.364} C_VEL
LIN {X 0,Y 143.641,Z 509.634,A -85,B 0,C 180,E1 -26254.652,E2 -26254.652} C_VEL
LIN {X 0,Y 144.002,Z 505.386,A -85,B 0,C 180,E1 -26258.015,E2 -26258.015} C_VEL
LIN {X 0,Y 143.919,Z 501.427,A -85,B 0,C 180,E1 -26261.494,E2 -26261.494} C_VEL
LIN {X 0,Y 143.725,Z 498.409,A -85,B 0,C 180,E1 -26264.399,E2 -26264.399} C_VEL
LIN {X 0,Y 143.108,Z 494.251,A -85,B 0,C 180,E1 -26269.168,E2 -26269.168} C_VEL
LIN {X 0,Y 142.853,Z 492.472,A -85,B 0,C 180,E1 -26271.513,E2 -26271.513} C_VEL
LIN {X 0,Y 142.316,Z 489.249,A -85,B 0,C 180,E1 -26277.17,E2 -26277.17} C_VEL
LIN {X 0,Y 142.064,Z 488.269,A -85,B 0,C 180,E1 -26280.001,E2 -26280.001} C_VEL
LIN {X 0,Y 141.683,Z 487.988,A -85,B 0,C 180,E1 -26282.844,E2 -26282.844} C_VEL
LIN {X 0,Y 141.375,Z 488.356,A -85,B 0,C 180,E1 -26288.577,E2 -26288.577} C_VEL
LIN {X 0,Y 141.688,Z 490.006,A -85,B 0,C 180,E1 -26294.36,E2 -26294.36} C_VEL
LIN {X 0,Y 142.219,Z 493.441,A -85,B 0,C 180,E1 -26300.238,E2 -26300.238} C_VEL
LIN {X 0,Y 142.45,Z 494.447,A -85,B 0,C 180,E1 -26301.718,E2 -26301.718} C_VEL
LIN {X 0,Y 142.917,Z 498.565,A -85,B 0,C 180,E1 -26306.269,E2 -26306.269} C_VEL
LIN {X 0,Y 143.248,Z 503.189,A -85,B 0,C 180,E1 -26310.511,E2 -26310.511} C_VEL
LIN {X 0,Y 143.3,Z 507.906,A -85,B 0,C 180,E1 -26314.332,E2 -26314.332} C_VEL
LIN {X 0,Y 143.127,Z 511.306,A -85,B 0,C 180,E1 -26316.873,E2 -26316.873} C_VEL
LIN {X 0,Y 142.844,Z 513.034,A -85,B 0,C 180,E1 -26318.075,E2 -26318.075} C_VEL
LIN {X 0,Y 140.474,Z 518.773,A -85,B 0,C 180,E1 -26321.37,E2 -26321.37} C_VEL
LIN {X 0,Y 137.647,Z 523.818,A -85,B 0,C 180,E1 -26324.372,E2 -26324.372} C_VEL
LIN {X 0,Y 131.011,Z 530.415,A -85,B 0,C 180,E1 -26327.891,E2 -26327.891} C_VEL
LIN {X 0,Y 124.48,Z 536.192,A -85,B 0,C 180,E1 -26332.226,E2 -26332.226} C_VEL
LIN {X 0,Y 117.971,Z 541.014,A -85,B 0,C 180,E1 -26337.577,E2 -26337.577} C_VEL
LIN {X 0,Y 112.246,Z 544.567,A -85,B 0,C 180,E1 -26344.005,E2 -26344.005} C_VEL
LIN {X 0,Y 109.943,Z 545.728,A -85,B 0,C 180,E1 -26347.446,E2 -26347.446} C_VEL
LIN {X 0,Y 106.82,Z 546.852,A -85,B 0,C 180,E1 -26354.741,E2 -26354.741} C_VEL
LIN {X 0,Y 105.296,Z 546.475,A -85,B 0,C 180,E1 -26362.328,E2 -26362.328} C_VEL
LIN {X 0,Y 105.18,Z 545.674,A -85,B 0,C 180,E1 -26366.168,E2 -26366.168} C_VEL
LIN {X 0,Y 105.234,Z 544.466,A -85,B 0,C 180,E1 -26369.999,E2 -26369.999} C_VEL
LIN {X 0,Y 105.176,Z 541.832,A -85,B 0,C 180,E1 -26375.752,E2 -26375.752} C_VEL
LIN {X 0,Y 105.821,Z 538.154,A -85,B 0,C 180,E1 -26381.492,E2 -26381.492} C_VEL
LIN {X 0,Y 107.181,Z 533.325,A -85,B 0,C 180,E1 -26387.161,E2 -26387.161} C_VEL
LIN {X 0,Y 109.589,Z 527.22,A -85,B 0,C 180,E1 -26392.629,E2 -26392.629} C_VEL
LIN {X 0,Y 112.803,Z 519.599,A -85,B 0,C 180,E1 -26397.856,E2 -26397.856} C_VEL
LIN {X 0,Y 116.069,Z 511.706,A -85,B 0,C 180,E1 -26402.036,E2 -26402.036} C_VEL
LIN {X 0,Y 118.709,Z 505.291,A -85,B 0,C 180,E1 -26404.737,E2 -26404.737} C_VEL
LIN {X 0,Y 120.341,Z 494.959,A -85,B 0,C 180,E1 -26408.887,E2 -26408.887} C_VEL
LIN {X 0,Y 121.188,Z 485.962,A -85,B 0,C 180,E1 -26411.987,E2 -26411.987} C_VEL
LIN {X 0,Y 121.303,Z 475.061,A -85,B 0,C 180,E1 -26415.403,E2 -26415.403} C_VEL
LIN {X 0,Y 120.929,Z 470.014,A -85,B 0,C 180,E1 -26416.931,E2 -26416.931} C_VEL
LIN {X 0,Y 118.366,Z 462.245,A -85,B 0,C 180,E1 -26419.923,E2 -26419.923} C_VEL
LIN {X 0,Y 114.952,Z 454.429,A -85,B 0,C 180,E1 -26423.271,E2 -26423.271} C_VEL
LIN {X 0,Y 113.272,Z 451.063,A -85,B 0,C 180,E1 -26424.84,E2 -26424.84} C_VEL
LIN {X 0,Y 111.281,Z 447.866,A -85,B 0,C 180,E1 -26426.602,E2 -26426.602} C_VEL
LIN {X 0,Y 110.513,Z 446.82,A -85,B 0,C 180,E1 -26427.268,E2 -26427.268} C_VEL
LIN {X 0,Y 108.652,Z 444.642,A -85,B 0,C 180,E1 -26428.837,E2 -26428.837} C_VEL
LIN {X 0,Y 107.809,Z 442.037,A -85,B 0,C 180,E1 -26429.924,E2 -26429.924} C_VEL
LIN {X 0,Y 107.908,Z 442.043,A -85,B 0,C 180,E1 -26436.996,E2 -26436.996} C_VEL
LIN {X 0,Y 108.029,Z 441.988,A -85,B 0,C 180,E1 -26444.916,E2 -26444.916} C_VEL
LIN {X 0,Y 108.3,Z 441.992,A -85,B 0,C 180,E1 -26448.773,E2 -26448.773} C_VEL
LIN {X 0,Y 108.453,Z 441.924,A -85,B 0,C 180,E1 -26456.284,E2 -26456.284} C_VEL
LIN {X 0,Y 108.918,Z 441.887,A -85,B 0,C 180,E1 -26459.999,E2 -26459.999} C_VEL
LIN {X 0,Y 108.325,Z 441.968,A -85,B 0,C 180,E1 -26467.455,E2 -26467.455} C_VEL
LIN {X 0,Y 108.196,Z 441.96,A -85,B 0,C 180,E1 -26473.015,E2 -26473.015} C_VEL
LIN {X 0,Y 107.901,Z 442.044,A -85,B 0,C 180,E1 -26479.005,E2 -26479.005} C_VEL
LIN {X 0,Y 107.853,Z 442.046,A -85,B 0,C 180,E1 -26484.182,E2 -26484.182} C_VEL
LIN {X 0,Y 107.73,Z 442.057,A -85,B 0,C 180,E1 -26487.534,E2 -26487.534} C_VEL
LIN {X 0,Y 106.971,Z 442.149,A -85,B 0,C 180,E1 -26489.6,E2 -26489.6} C_VEL
LIN {X 0,Y 104.07,Z 442.521,A -85,B 0,C 180,E1 -26492.876,E2 -26492.876} C_VEL
LIN {X 0,Y 101.252,Z 442.862,A -85,B 0,C 180,E1 -26496.332,E2 -26496.332} C_VEL
LIN {X 0,Y 100.701,Z 442.938,A -85,B 0,C 180,E1 -26498.594,E2 -26498.594} C_VEL
LIN {X 0,Y 100.755,Z 443.144,A -85,B 0,C 180,E1 -26499.357,E2 -26499.357} C_VEL
LIN {X 0,Y 101.597,Z 445.577,A -85,B 0,C 180,E1 -26500.725,E2 -26500.725} C_VEL
LIN {X 0,Y 103.673,Z 447.857,A -85,B 0,C 180,E1 -26503.005,E2 -26503.005} C_VEL
LIN {X 0,Y 104.357,Z 448.887,A -85,B 0,C 180,E1 -26503.779,E2 -26503.779} C_VEL
LIN {X 0,Y 106.301,Z 452.026,A -85,B 0,C 180,E1 -26506.013,E2 -26506.013} C_VEL
LIN {X 0,Y 107.332,Z 453.587,A -85,B 0,C 180,E1 -26507.099,E2 -26507.099} C_VEL
LIN {X 0,Y 110.003,Z 458.386,A -85,B 0,C 180,E1 -26510.055,E2 -26510.055} C_VEL
LIN {X 0,Y 113.74,Z 466.016,A -85,B 0,C 180,E1 -26514.27,E2 -26514.27} C_VEL
LIN {X 0,Y 115.884,Z 471.305,A -85,B 0,C 180,E1 -26516.921,E2 -26516.921} C_VEL
LIN {X 0,Y 116.417,Z 474.148,A -85,B 0,C 180,E1 -26518.074,E2 -26518.074} C_VEL
LIN {X 0,Y 116.687,Z 483.688,A -85,B 0,C 180,E1 -26521.687,E2 -26521.687} C_VEL
LIN {X 0,Y 116.288,Z 491.86,A -85,B 0,C 180,E1 -26525.031,E2 -26525.031} C_VEL
LIN {X 0,Y 112.195,Z 502.1,A -85,B 0,C 180,E1 -26528.89,E2 -26528.89} C_VEL
LIN {X 0,Y 108.361,Z 510.538,A -85,B 0,C 180,E1 -26533.032,E2 -26533.032} C_VEL
LIN {X 0,Y 104.491,Z 518.788,A -85,B 0,C 180,E1 -26538.36,E2 -26538.36} C_VEL
LIN {X 0,Y 101.604,Z 525.416,A -85,B 0,C 180,E1 -26544.045,E2 -26544.045} C_VEL
LIN {X 0,Y 99.561,Z 530.704,A -85,B 0,C 180,E1 -26550.001,E2 -26550.001} C_VEL
LIN {X 0,Y 98.218,Z 534.834,A -85,B 0,C 180,E1 -26556.162,E2 -26556.162} C_VEL
LIN {X 0,Y 97.586,Z 537.909,A -85,B 0,C 180,E1 -26562.478,E2 -26562.478} C_VEL
LIN {X 0,Y 97.695,Z 539.394,A -85,B 0,C 180,E1 -26566.724,E2 -26566.724} C_VEL
LIN {X 0,Y 98.359,Z 540.605,A -85,B 0,C 180,E1 -26571.741,E2 -26571.741} C_VEL
LIN {X 0,Y 100.385,Z 541.351,A -85,B 0,C 180,E1 -26579.346,E2 -26579.346} C_VEL
LIN {X 0,Y 103.121,Z 540.929,A -85,B 0,C 180,E1 -26585.132,E2 -26585.132} C_VEL
LIN {X 0,Y 107.034,Z 539.481,A -85,B 0,C 180,E1 -26591.042,E2 -26591.042} C_VEL
LIN {X 0,Y 111.599,Z 537.152,A -85,B 0,C 180,E1 -26596.154,E2 -26596.154} C_VEL
LIN {X 0,Y 117.376,Z 533.591,A -85,B 0,C 180,E1 -26601.113,E2 -26601.113} C_VEL
LIN {X 0,Y 124.184,Z 528.532,A -85,B 0,C 180,E1 -26605.788,E2 -26605.788} C_VEL
LIN {X 0,Y 131.864,Z 521.809,A -85,B 0,C 180,E1 -26610.006,E2 -26610.006} C_VEL
LIN {X 0,Y 135.59,Z 518.13,A -85,B 0,C 180,E1 -26611.781,E2 -26611.781} C_VEL
LIN {X 0,Y 136.782,Z 515.935,A -85,B 0,C 180,E1 -26613.283,E2 -26613.283} C_VEL
LIN {X 0,Y 138.029,Z 511.96,A -85,B 0,C 180,E1 -26616.419,E2 -26616.419} C_VEL
LIN {X 0,Y 138.428,Z 508.872,A -85,B 0,C 180,E1 -26619.183,E2 -26619.183} C_VEL
LIN {X 0,Y 138.658,Z 504.584,A -85,B 0,C 180,E1 -26623.356,E2 -26623.356} C_VEL
LIN {X 0,Y 138.429,Z 500.395,A -85,B 0,C 180,E1 -26628.283,E2 -26628.283} C_VEL
LIN {X 0,Y 138.281,Z 498.292,A -85,B 0,C 180,E1 -26631.23,E2 -26631.23} C_VEL
LIN {X 0,Y 138.132,Z 496.51,A -85,B 0,C 180,E1 -26634.16,E2 -26634.16} C_VEL
LIN {X 0,Y 138.056,Z 495.054,A -85,B 0,C 180,E1 -26637.083,E2 -26637.083} C_VEL
LIN {X 0,Y 137.906,Z 494.042,A -85,B 0,C 180,E1 -26640.001,E2 -26640.001} C_VEL
LIN {X 0,Y 137.555,Z 493.771,A -85,B 0,C 180,E1 -26642.929,E2 -26642.929} C_VEL
LIN {X 0,Y 137.234,Z 494.224,A -85,B 0,C 180,E1 -26648.838,E2 -26648.838} C_VEL
LIN {X 0,Y 137.41,Z 495.506,A -85,B 0,C 180,E1 -26653.647,E2 -26653.647} C_VEL
LIN {X 0,Y 137.524,Z 497.651,A -85,B 0,C 180,E1 -26657.856,E2 -26657.856} C_VEL
LIN {X 0,Y 137.795,Z 499.485,A -85,B 0,C 180,E1 -26660.918,E2 -26660.918} C_VEL
LIN {X 0,Y 137.951,Z 503.409,A -85,B 0,C 180,E1 -26665.661,E2 -26665.661} C_VEL
LIN {X 0,Y 137.927,Z 508.46,A -85,B 0,C 180,E1 -26670.634,E2 -26670.634} C_VEL
LIN {X 0,Y 137.485,Z 513.713,A -85,B 0,C 180,E1 -26675.126,E2 -26675.126} C_VEL
LIN {X 0,Y 136.81,Z 516.503,A -85,B 0,C 180,E1 -26677.23,E2 -26677.23} C_VEL
LIN {X 0,Y 134.076,Z 521.805,A -85,B 0,C 180,E1 -26680.531,E2 -26680.531} C_VEL
LIN {X 0,Y 132.621,Z 524.186,A -85,B 0,C 180,E1 -26682.107,E2 -26682.107} C_VEL
LIN {X 0,Y 129.269,Z 527.595,A -85,B 0,C 180,E1 -26683.916,E2 -26683.916} C_VEL
LIN {X 0,Y 123.648,Z 532.517,A -85,B 0,C 180,E1 -26686.995,E2 -26686.995} C_VEL
LIN {X 0,Y 116.826,Z 537.843,A -85,B 0,C 180,E1 -26691.638,E2 -26691.638} C_VEL
LIN {X 0,Y 112.045,Z 541.043,A -85,B 0,C 180,E1 -26695.631,E2 -26695.631} C_VEL
LIN {X 0,Y 105.896,Z 544.512,A -85,B 0,C 180,E1 -26702.318,E2 -26702.318} C_VEL
LIN {X 0,Y 101.434,Z 546.323,A -85,B 0,C 180,E1 -26709.73,E2 -26709.73} C_VEL
LIN {X 0,Y 98.909,Z 546.632,A -85,B 0,C 180,E1 -26717.691,E2 -26717.691} C_VEL
LIN {X 0,Y 98.263,Z 546.193,A -85,B 0,C 180,E1 -26721.775,E2 -26721.775} C_VEL
LIN {X 0,Y 98.091,Z 545.348,A -85,B 0,C 180,E1 -26725.891,E2 -26725.891} C_VEL
LIN {X 0,Y 98.146,Z 544.107,A -85,B 0,C 180,E1 -26729.999,E2 -26729.999} C_VEL
LIN {X 0,Y 98.1,Z 541.398,A -85,B 0,C 180,E1 -26736.168,E2 -26736.168} C_VEL
LIN {X 0,Y 98.861,Z 537.643,A -85,B 0,C 180,E1 -26742.313,E2 -26742.313} C_VEL
LIN {X 0,Y 100.362,Z 532.727,A -85,B 0,C 180,E1 -26748.367,E2 -26748.367} C_VEL
LIN {X 0,Y 103.011,Z 526.53,A -85,B 0,C 180,E1 -26754.163,E2 -26754.163} C_VEL
LIN {X 0,Y 106.544,Z 518.789,A -85,B 0,C 180,E1 -26759.65,E2 -26759.65} C_VEL
LIN {X 0,Y 108.993,Z 512.973,A -85,B 0,C 180,E1 -26762.926,E2 -26762.926} C_VEL
LIN {X 0,Y 112.071,Z 506.216,A -85,B 0,C 180,E1 -26766.007,E2 -26766.007} C_VEL
LIN {X 0,Y 113.808,Z 497.379,A -85,B 0,C 180,E1 -26769.841,E2 -26769.841} C_VEL
LIN {X 0,Y 114.996,Z 488.254,A -85,B 0,C 180,E1 -26773.289,E2 -26773.289} C_VEL
LIN {X 0,Y 115.487,Z 476.28,A -85,B 0,C 180,E1 -26777.33,E2 -26777.33} C_VEL
LIN {X 0,Y 115.191,Z 472.643,A -85,B 0,C 180,E1 -26778.581,E2 -26778.581} C_VEL
LIN {X 0,Y 112.374,Z 463.844,A -85,B 0,C 180,E1 -26782.426,E2 -26782.426} C_VEL
LIN {X 0,Y 109.252,Z 456.461,A -85,B 0,C 180,E1 -26786.023,E2 -26786.023} C_VEL
LIN {X 0,Y 106.678,Z 452.38,A -85,B 0,C 180,E1 -26788.65,E2 -26788.65} C_VEL
LIN {X 0,Y 104.671,Z 449.31,A -85,B 0,C 180,E1 -26790.756,E2 -26790.756} C_VEL
LIN {X 0,Y 104.042,Z 448.064,A -85,B 0,C 180,E1 -26791.52,E2 -26791.52} C_VEL
LIN {X 0,Y 101.793,Z 445.889,A -85,B 0,C 180,E1 -26793.847,E2 -26793.847} C_VEL
LIN {X 0,Y 100.852,Z 443.395,A -85,B 0,C 180,E1 -26795.205,E2 -26795.205} C_VEL
LIN {X 0,Y 100.79,Z 442.916,A -85,B 0,C 180,E1 -26795.465,E2 -26795.465} C_VEL
LIN {X 0,Y 100.809,Z 442.91,A -85,B 0,C 180,E1 -26799.599,E2 -26799.599} C_VEL
LIN {X 0,Y 101.194,Z 442.871,A -85,B 0,C 180,E1 -26807.973,E2 -26807.973} C_VEL
LIN {X 0,Y 101.272,Z 442.857,A -85,B 0,C 180,E1 -26812.021,E2 -26812.021} C_VEL
LIN {X 0,Y 101.846,Z 442.764,A -85,B 0,C 180,E1 -26819.999,E2 -26819.999} C_VEL
LIN {X 0,Y 101.264,Z 442.837,A -85,B 0,C 180,E1 -26827.978,E2 -26827.978} C_VEL
LIN {X 0,Y 101.121,Z 442.842,A -85,B 0,C 180,E1 -26833.351,E2 -26833.351} C_VEL
LIN {X 0,Y 100.813,Z 442.92,A -85,B 0,C 180,E1 -26840.399,E2 -26840.399} C_VEL
LIN {X 0,Y 100.771,Z 442.932,A -85,B 0,C 180,E1 -26844.959,E2 -26844.959} C_VEL
LIN {X 0,Y 100.706,Z 442.938,A -85,B 0,C 180,E1 -26853.132,E2 -26853.132} C_VEL
LIN {X 0,Y 100.701,Z 442.938,A -85,B 0,C 180,E1 -26858.594,E2 -26858.594} C_VEL
LIN {X 0,Y 101.476,Z 443.446,A -85,B 0,C 180,E1 -26860.063,E2 -26860.063} C_VEL
LIN {X 0,Y 102.903,Z 445.236,A -85,B 0,C 180,E1 -26861.757,E2 -26861.757} C_VEL
LIN {X 0,Y 104.202,Z 448.625,A -85,B 0,C 180,E1 -26863.596,E2 -26863.596} C_VEL
LIN {X 0,Y 105.299,Z 455.531,A -85,B 0,C 180,E1 -26866.116,E2 -26866.116} C_VEL
LIN {X 0,Y 105.837,Z 462.687,A -85,B 0,C 180,E1 -26868.788,E2 -26868.788} C_VEL
LIN {X 0,Y 106.658,Z 465.736,A -85,B 0,C 180,E1 -26870.37,E2 -26870.37} C_VEL
LIN {X 0,Y 109.755,Z 473.476,A -85,B 0,C 180,E1 -26874.811,E2 -26874.811} C_VEL
LIN {X 0,Y 110.559,Z 476.066,A -85,B 0,C 180,E1 -26876.175,E2 -26876.175} C_VEL
LIN {X 0,Y 110.668,Z 484.098,A -85,B 0,C 180,E1 -26879.468,E2 -26879.468} C_VEL
LIN {X 0,Y 110.021,Z 493.207,A -85,B 0,C 180,E1 -26883.44,E2 -26883.44} C_VEL
LIN {X 0,Y 105.57,Z 503.303,A -85,B 0,C 180,E1 -26887.495,E2 -26887.495} C_VEL
LIN {X 0,Y 101.545,Z 511.578,A -85,B 0,C 180,E1 -26891.855,E2 -26891.855} C_VEL
LIN {X 0,Y 97.49,Z 519.686,A -85,B 0,C 180,E1 -26897.511,E2 -26897.511} C_VEL
LIN {X 0,Y 94.514,Z 526.178,A -85,B 0,C 180,E1 -26903.597,E2 -26903.597} C_VEL
LIN {X 0,Y 92.402,Z 531.338,A -85,B 0,C 180,E1 -26910.001,E2 -26910.001} C_VEL
LIN {X 0,Y 91.032,Z 535.364,A -85,B 0,C 180,E1 -26916.651,E2 -26916.651} C_VEL
LIN {X 0,Y 90.464,Z 538.351,A -85,B 0,C 180,E1 -26923.478,E2 -26923.478} C_VEL
LIN {X 0,Y 90.693,Z 539.764,A -85,B 0,C 180,E1 -26928.058,E2 -26928.058} C_VEL
LIN {X 0,Y 91.394,Z 540.783,A -85,B 0,C 180,E1 -26932.667,E2 -26932.667} C_VEL
LIN {X 0,Y 92.419,Z 541.387,A -85,B 0,C 180,E1 -26937.147,E2 -26937.147} C_VEL
LIN {X 0,Y 93.995,Z 541.543,A -85,B 0,C 180,E1 -26941.56,E2 -26941.56} C_VEL
LIN {X 0,Y 96.698,Z 541.157,A -85,B 0,C 180,E1 -26946.921,E2 -26946.921} C_VEL
LIN {X 0,Y 101.521,Z 539.513,A -85,B 0,C 180,E1 -26953.81,E2 -26953.81} C_VEL
LIN {X 0,Y 105.905,Z 537.442,A -85,B 0,C 180,E1 -26958.425,E2 -26958.425} C_VEL
LIN {X 0,Y 112.839,Z 533.429,A -85,B 0,C 180,E1 -26964.065,E2 -26964.065} C_VEL
LIN {X 0,Y 119.902,Z 528.432,A -85,B 0,C 180,E1 -26968.589,E2 -26968.589} C_VEL
LIN {X 0,Y 128.325,Z 521.41,A -85,B 0,C 180,E1 -26972.857,E2 -26972.857} C_VEL
LIN {X 0,Y 129.605,Z 520.211,A -85,B 0,C 180,E1 -26973.451,E2 -26973.451} C_VEL
LIN {X 0,Y 130.896,Z 518.515,A -85,B 0,C 180,E1 -26974.563,E2 -26974.563} C_VEL
LIN {X 0,Y 131.833,Z 516.321,A -85,B 0,C 180,E1 -26976.439,E2 -26976.439} C_VEL
LIN {X 0,Y 132.71,Z 512.774,A -85,B 0,C 180,E1 -26979.866,E2 -26979.866} C_VEL
LIN {X 0,Y 133.121,Z 509.748,A -85,B 0,C 180,E1 -26983.11,E2 -26983.11} C_VEL
LIN {X 0,Y 133.333,Z 507.086,A -85,B 0,C 180,E1 -26986.279,E2 -26986.279} C_VEL
LIN {X 0,Y 133.395,Z 503.823,A -85,B 0,C 180,E1 -26990.906,E2 -26990.906} C_VEL
LIN {X 0,Y 133.378,Z 502.059,A -85,B 0,C 180,E1 -26993.951,E2 -26993.951} C_VEL
LIN {X 0,Y 133.434,Z 500.603,A -85,B 0,C 180,E1 -26996.981,E2 -26996.981} C_VEL
LIN {X 0,Y 133.439,Z 499.586,A -85,B 0,C 180,E1 -27000.001,E2 -27000.001} C_VEL
LIN {X 0,Y 133.123,Z 499.323,A -85,B 0,C 180,E1 -27003.027,E2 -27003.027} C_VEL
LIN {X 0,Y 132.79,Z 499.851,A -85,B 0,C 180,E1 -27009.136,E2 -27009.136} C_VEL
LIN {X 0,Y 132.836,Z 500.581,A -85,B 0,C 180,E1 -27012.218,E2 -27012.218} C_VEL
LIN {X 0,Y 132.793,Z 503.009,A -85,B 0,C 180,E1 -27017.705,E2 -27017.705} C_VEL
LIN {X 0,Y 132.902,Z 504.341,A -85,B 0,C 180,E1 -27020.105,E2 -27020.105} C_VEL
LIN {X 0,Y 132.766,Z 508.055,A -85,B 0,C 180,E1 -27025.055,E2 -27025.055} C_VEL
LIN {X 0,Y 132.364,Z 512.783,A -85,B 0,C 180,E1 -27030.122,E2 -27030.122} C_VEL
LIN {X 0,Y 131.673,Z 516.997,A -85,B 0,C 180,E1 -27034.086,E2 -27034.086} C_VEL
LIN {X 0,Y 131.356,Z 518.317,A -85,B 0,C 180,E1 -27035.229,E2 -27035.229} C_VEL
LIN {X 0,Y 130.136,Z 520.735,A -85,B 0,C 180,E1 -27036.97,E2 -27036.97} C_VEL
LIN {X 0,Y 126.846,Z 525.683,A -85,B 0,C 180,E1 -27040.375,E2 -27040.375} C_VEL
LIN {X 0,Y 118.545,Z 532.725,A -85,B 0,C 180,E1 -27044.649,E2 -27044.649} C_VEL
LIN {X 0,Y 112.442,Z 537.209,A -85,B 0,C 180,E1 -27048.595,E2 -27048.595} C_VEL
LIN {X 0,Y 106.265,Z 541.081,A -85,B 0,C 180,E1 -27053.471,E2 -27053.471} C_VEL
LIN {X 0,Y 102.732,Z 542.979,A -85,B 0,C 180,E1 -27056.819,E2 -27056.819} C_VEL
LIN {X 0,Y 99.653,Z 544.442,A -85,B 0,C 180,E1 -27060.418,E2 -27060.418} C_VEL
LIN {X 0,Y 94.771,Z 546.171,A -85,B 0,C 180,E1 -27068.235,E2 -27068.235} C_VEL
LIN {X 0,Y 91.954,Z 546.398,A -85,B 0,C 180,E1 -27076.744,E2 -27076.744} C_VEL
LIN {X 0,Y 91.004,Z 545.023,A -85,B 0,C 180,E1 -27085.57,E2 -27085.57} C_VEL
LIN {X 0,Y 91.05,Z 543.747,A -85,B 0,C 180,E1 -27089.999,E2 -27089.999} C_VEL
LIN {X 0,Y 91.051,Z 540.965,A -85,B 0,C 180,E1 -27096.648,E2 -27096.648} C_VEL
LIN {X 0,Y 91.892,Z 537.13,A -85,B 0,C 180,E1 -27103.263,E2 -27103.263} C_VEL
LIN {X 0,Y 93.609,Z 532.131,A -85,B 0,C 180,E1 -27109.745,E2 -27109.745} C_VEL
LIN {X 0,Y 96.535,Z 525.842,A -85,B 0,C 180,E1 -27115.9,E2 -27115.9} C_VEL
LIN {X 0,Y 100.376,Z 517.941,A -85,B 0,C 180,E1 -27121.675,E2 -27121.675} C_VEL
LIN {X 0,Y 102.807,Z 512.621,A -85,B 0,C 180,E1 -27124.784,E2 -27124.784} C_VEL
LIN {X 0,Y 105.864,Z 506.141,A -85,B 0,C 180,E1 -27127.883,E2 -27127.883} C_VEL
LIN {X 0,Y 107.895,Z 496.47,A -85,B 0,C 180,E1 -27132.299,E2 -27132.299} C_VEL
LIN {X 0,Y 109.197,Z 486.976,A -85,B 0,C 180,E1 -27136.054,E2 -27136.054} C_VEL
LIN {X 0,Y 109.763,Z 477.15,A -85,B 0,C 180,E1 -27139.582,E2 -27139.582} C_VEL
LIN {X 0,Y 108.36,Z 471.041,A -85,B 0,C 180,E1 -27142.375,E2 -27142.375} C_VEL
LIN {X 0,Y 105.471,Z 462.877,A -85,B 0,C 180,E1 -27146.651,E2 -27146.651} C_VEL
LIN {X 0,Y 103.372,Z 458.576,A -85,B 0,C 180,E1 -27149.342,E2 -27149.342} C_VEL
LIN {X 0,Y 101.049,Z 454.992,A -85,B 0,C 180,E1 -27152.141,E2 -27152.141} C_VEL
LIN {X 0,Y 100.452,Z 453.919,A -85,B 0,C 180,E1 -27152.949,E2 -27152.949} C_VEL
LIN {X 0,Y 98.281,Z 451.123,A -85,B 0,C 180,E1 -27155.726,E2 -27155.726} C_VEL
LIN {X 0,Y 97.334,Z 449.1,A -85,B 0,C 180,E1 -27157.238,E2 -27157.238} C_VEL
LIN {X 0,Y 94.962,Z 446.932,A -85,B 0,C 180,E1 -27160.546,E2 -27160.546} C_VEL
LIN {X 0,Y 93.964,Z 444.725,A -85,B 0,C 180,E1 -27162.45,E2 -27162.45} C_VEL
LIN {X 0,Y 93.806,Z 443.753,A -85,B 0,C 180,E1 -27163.015,E2 -27163.015} C_VEL
LIN {X 0,Y 94.08,Z 443.742,A -85,B 0,C 180,E1 -27167.049,E2 -27167.049} C_VEL
LIN {X 0,Y 94.205,Z 443.743,A -85,B 0,C 180,E1 -27171.418,E2 -27171.418} C_VEL
LIN {X 0,Y 94.776,Z 443.642,A -85,B 0,C 180,E1 -27179.999,E2 -27179.999} C_VEL
LIN {X 0,Y 94.197,Z 443.708,A -85,B 0,C 180,E1 -27188.581,E2 -27188.581} C_VEL
LIN {X 0,Y 94.039,Z 443.725,A -85,B 0,C 180,E1 -27193.708,E2 -27193.708} C_VEL
LIN {X 0,Y 93.689,Z 443.802,A -85,B 0,C 180,E1 -27202.028,E2 -27202.028} C_VEL
LIN {X 0,Y 93.618,Z 443.819,A -85,B 0,C 180,E1 -27206.77,E2 -27206.77} C_VEL
LIN {X 0,Y 93.604,Z 443.907,A -85,B 0,C 180,E1 -27211.548,E2 -27211.548} C_VEL
LIN {X 0,Y 94.634,Z 446.611,A -85,B 0,C 180,E1 -27213.818,E2 -27213.818} C_VEL
LIN {X 0,Y 96.677,Z 448.84,A -85,B 0,C 180,E1 -27216.851,E2 -27216.851} C_VEL
LIN {X 0,Y 97.523,Z 449.461,A -85,B 0,C 180,E1 -27217.934,E2 -27217.934} C_VEL
LIN {X 0,Y 99.198,Z 452.762,A -85,B 0,C 180,E1 -27220.62,E2 -27220.62} C_VEL
LIN {X 0,Y 100.637,Z 454.415,A -85,B 0,C 180,E1 -27222.376,E2 -27222.376} C_VEL
LIN {X 0,Y 104.84,Z 461.789,A -85,B 0,C 180,E1 -27227.908,E2 -27227.908} C_VEL
LIN {X 0,Y 106.658,Z 465.736,A -85,B 0,C 180,E1 -27230.37,E2 -27230.37} C_VEL
LIN {X 0,Y 107.379,Z 469.145,A -85,B 0,C 180,E1 -27231.968,E2 -27231.968} C_VEL
LIN {X 0,Y 106.859,Z 474.252,A -85,B 0,C 180,E1 -27233.606,E2 -27233.606} C_VEL
LIN {X 0,Y 104.944,Z 482.495,A -85,B 0,C 180,E1 -27236.147,E2 -27236.147} C_VEL
LIN {X 0,Y 104.84,Z 483.585,A -85,B 0,C 180,E1 -27236.593,E2 -27236.593} C_VEL
LIN {X 0,Y 103.99,Z 493.531,A -85,B 0,C 180,E1 -27241.216,E2 -27241.216} C_VEL
LIN {X 0,Y 103.256,Z 495.638,A -85,B 0,C 180,E1 -27242.101,E2 -27242.101} C_VEL
LIN {X 0,Y 98.14,Z 506.243,A -85,B 0,C 180,E1 -27246.806,E2 -27246.806} C_VEL
LIN {X 0,Y 93.29,Z 515.411,A -85,B 0,C 180,E1 -27252.463,E2 -27252.463} C_VEL
LIN {X 0,Y 89.373,Z 522.796,A -85,B 0,C 180,E1 -27258.663,E2 -27258.663} C_VEL
LIN {X 0,Y 86.534,Z 528.709,A -85,B 0,C 180,E1 -27265.342,E2 -27265.342} C_VEL
LIN {X 0,Y 84.477,Z 533.89,A -85,B 0,C 180,E1 -27273.32,E2 -27273.32} C_VEL
LIN {X 0,Y 83.539,Z 536.961,A -85,B 0,C 180,E1 -27279.687,E2 -27279.687} C_VEL
LIN {X 0,Y 83.368,Z 538.76,A -85,B 0,C 180,E1 -27284.65,E2 -27284.65} C_VEL
LIN {X 0,Y 84.429,Z 540.95,A -85,B 0,C 180,E1 -27293.703,E2 -27293.703} C_VEL
LIN {X 0,Y 85.904,Z 541.637,A -85,B 0,C 180,E1 -27299.398,E2 -27299.398} C_VEL
LIN {X 0,Y 87.754,Z 541.733,A -85,B 0,C 180,E1 -27304.098,E2 -27304.098} C_VEL
LIN {X 0,Y 90.333,Z 541.391,A -85,B 0,C 180,E1 -27308.923,E2 -27308.923} C_VEL
LIN {X 0,Y 92.974,Z 540.712,A -85,B 0,C 180,E1 -27312.869,E2 -27312.869} C_VEL
LIN {X 0,Y 96.28,Z 539.524,A -85,B 0,C 180,E1 -27316.883,E2 -27316.883} C_VEL
LIN {X 0,Y 100.437,Z 537.718,A -85,B 0,C 180,E1 -27320.968,E2 -27320.968} C_VEL
LIN {X 0,Y 106.358,Z 534.592,A -85,B 0,C 180,E1 -27325.688,E2 -27325.688} C_VEL
LIN {X 0,Y 113.768,Z 529.893,A -85,B 0,C 180,E1 -27330.384,E2 -27330.384} C_VEL
LIN {X 0,Y 122.403,Z 523.287,A -85,B 0,C 180,E1 -27334.731,E2 -27334.731} C_VEL
LIN {X 0,Y 125.072,Z 520.854,A -85,B 0,C 180,E1 -27336.109,E2 -27336.109} C_VEL
LIN {X 0,Y 126.372,Z 518.106,A -85,B 0,C 180,E1 -27338.811,E2 -27338.811} C_VEL
LIN {X 0,Y 127.238,Z 515.12,A -85,B 0,C 180,E1 -27342.142,E2 -27342.142} C_VEL
LIN {X 0,Y 127.94,Z 511.138,A -85,B 0,C 180,E1 -27347.307,E2 -27347.307} C_VEL
LIN {X 0,Y 128.161,Z 508.92,A -85,B 0,C 180,E1 -27350.773,E2 -27350.773} C_VEL
LIN {X 0,Y 128.315,Z 507.352,A -85,B 0,C 180,E1 -27353.712,E2 -27353.712} C_VEL
LIN {X 0,Y 128.495,Z 505.891,A -85,B 0,C 180,E1 -27356.865,E2 -27356.865} C_VEL
LIN {X 0,Y 128.636,Z 504.863,A -85,B 0,C 180,E1 -27360.001,E2 -27360.001} C_VEL
LIN {X 0,Y 128.375,Z 504.627,A -85,B 0,C 180,E1 -27363.139,E2 -27363.139} C_VEL
LIN {X 0,Y 128.052,Z 505.1,A -85,B 0,C 180,E1 -27368.922,E2 -27368.922} C_VEL
LIN {X 0,Y 127.952,Z 506.037,A -85,B 0,C 180,E1 -27372.692,E2 -27372.692} C_VEL
LIN {X 0,Y 127.826,Z 507.337,A -85,B 0,C 180,E1 -27375.957,E2 -27375.957} C_VEL
LIN {X 0,Y 127.803,Z 508.971,A -85,B 0,C 180,E1 -27379.266,E2 -27379.266} C_VEL
LIN {X 0,Y 127.379,Z 512.483,A -85,B 0,C 180,E1 -27384.445,E2 -27384.445} C_VEL
LIN {X 0,Y 126.757,Z 516.139,A -85,B 0,C 180,E1 -27388.809,E2 -27388.809} C_VEL
LIN {X 0,Y 125.767,Z 520.182,A -85,B 0,C 180,E1 -27393.049,E2 -27393.049} C_VEL
LIN {X 0,Y 124.815,Z 522.273,A -85,B 0,C 180,E1 -27394.891,E2 -27394.891} C_VEL
LIN {X 0,Y 121.135,Z 527.093,A -85,B 0,C 180,E1 -27398.442,E2 -27398.442} C_VEL
LIN {X 0,Y 113.66,Z 532.933,A -85,B 0,C 180,E1 -27402.098,E2 -27402.098} C_VEL
LIN {X 0,Y 106.629,Z 537.706,A -85,B 0,C 180,E1 -27406.472,E2 -27406.472} C_VEL
LIN {X 0,Y 100.653,Z 541.119,A -85,B 0,C 180,E1 -27411.067,E2 -27411.067} C_VEL
LIN {X 0,Y 96.853,Z 542.965,A -85,B 0,C 180,E1 -27414.513,E2 -27414.513} C_VEL
LIN {X 0,Y 90.603,Z 545.381,A -85,B 0,C 180,E1 -27422.263,E2 -27422.263} C_VEL
LIN {X 0,Y 86.361,Z 546.288,A -85,B 0,C 180,E1 -27431.002,E2 -27431.002} C_VEL
LIN {X 0,Y 84.206,Z 545.606,A -85,B 0,C 180,E1 -27440.39,E2 -27440.39} C_VEL
LIN {X 0,Y 83.915,Z 544.692,A -85,B 0,C 180,E1 -27445.195,E2 -27445.195} C_VEL
LIN {X 0,Y 83.947,Z 543.38,A -85,B 0,C 180,E1 -27449.999,E2 -27449.999} C_VEL
LIN {X 0,Y 83.986,Z 540.523,A -85,B 0,C 180,E1 -27457.21,E2 -27457.21} C_VEL
LIN {X 0,Y 84.965,Z 536.607,A -85,B 0,C 180,E1 -27464.367,E2 -27464.367} C_VEL
LIN {X 0,Y 87.374,Z 530.538,A -85,B 0,C 180,E1 -27472.461,E2 -27472.461} C_VEL
LIN {X 0,Y 90.804,Z 523.872,A -85,B 0,C 180,E1 -27478.928,E2 -27478.928} C_VEL
LIN {X 0,Y 94.327,Z 517.06,A -85,B 0,C 180,E1 -27483.971,E2 -27483.971} C_VEL
LIN {X 0,Y 97.108,Z 511.579,A -85,B 0,C 180,E1 -27487.239,E2 -27487.239} C_VEL
LIN {X 0,Y 99.412,Z 507.021,A -85,B 0,C 180,E1 -27489.512,E2 -27489.512} C_VEL
LIN {X 0,Y 101.581,Z 498.392,A -85,B 0,C 180,E1 -27493.775,E2 -27493.775} C_VEL
LIN {X 0,Y 103.188,Z 489.424,A -85,B 0,C 180,E1 -27497.64,E2 -27497.64} C_VEL
LIN {X 0,Y 104.076,Z 480.316,A -85,B 0,C 180,E1 -27501.225,E2 -27501.225} C_VEL
LIN {X 0,Y 103.78,Z 477.701,A -85,B 0,C 180,E1 -27502.447,E2 -27502.447} C_VEL
LIN {X 0,Y 101.298,Z 468.652,A -85,B 0,C 180,E1 -27507.472,E2 -27507.472} C_VEL
LIN {X 0,Y 99.454,Z 464.392,A -85,B 0,C 180,E1 -27510.352,E2 -27510.352} C_VEL
LIN {X 0,Y 96.881,Z 459.742,A -85,B 0,C 180,E1 -27514.198,E2 -27514.198} C_VEL
LIN {X 0,Y 94.827,Z 456.651,A -85,B 0,C 180,E1 -27517.389,E2 -27517.389} C_VEL
LIN {X 0,Y 94.138,Z 455.241,A -85,B 0,C 180,E1 -27518.656,E2 -27518.656} C_VEL
LIN {X 0,Y 91.824,Z 452.453,A -85,B 0,C 180,E1 -27522.603,E2 -27522.603} C_VEL
LIN {X 0,Y 90.995,Z 450.203,A -85,B 0,C 180,E1 -27524.703,E2 -27524.703} C_VEL
LIN {X 0,Y 88.25,Z 447.672,A -85,B 0,C 180,E1 -27530.834,E2 -27530.834} C_VEL
LIN {X 0,Y 87.31,Z 445.303,A -85,B 0,C 180,E1 -27534.659,E2 -27534.659} C_VEL
LIN {X 0,Y 87.25,Z 444.562,A -85,B 0,C 180,E1 -27535.668,E2 -27535.668} C_VEL
LIN {X 0,Y 87.706,Z 444.52,A -85,B 0,C 180,E1 -27539.999,E2 -27539.999} C_VEL
LIN {X 0,Y 87.105,Z 444.583,A -85,B 0,C 180,E1 -27549.286,E2 -27549.286} C_VEL
LIN {X 0,Y 86.948,Z 444.609,A -85,B 0,C 180,E1 -27554.087,E2 -27554.087} C_VEL
LIN {X 0,Y 86.729,Z 444.778,A -85,B 0,C 180,E1 -27557.841,E2 -27557.841} C_VEL
LIN {X 0,Y 87.295,Z 446.908,A -85,B 0,C 180,E1 -27561.24,E2 -27561.24} C_VEL
LIN {X 0,Y 89.767,Z 449.771,A -85,B 0,C 180,E1 -27568.017,E2 -27568.017} C_VEL
LIN {X 0,Y 90.934,Z 450.617,A -85,B 0,C 180,E1 -27570.316,E2 -27570.316} C_VEL
LIN {X 0,Y 92.552,Z 453.931,A -85,B 0,C 180,E1 -27573.989,E2 -27573.989} C_VEL
LIN {X 0,Y 94.224,Z 455.568,A -85,B 0,C 180,E1 -27576.633,E2 -27576.633} C_VEL
LIN {X 0,Y 95.69,Z 458.584,A -85,B 0,C 180,E1 -27579.408,E2 -27579.408} C_VEL
LIN {X 0,Y 96.694,Z 459.847,A -85,B 0,C 180,E1 -27580.854,E2 -27580.854} C_VEL
LIN {X 0,Y 100.299,Z 466.736,A -85,B 0,C 180,E1 -27586.576,E2 -27586.576} C_VEL
LIN {X 0,Y 103.249,Z 474.097,A -85,B 0,C 180,E1 -27591.519,E2 -27591.519} C_VEL
LIN {X 0,Y 104.787,Z 478.823,A -85,B 0,C 180,E1 -27594.41,E2 -27594.41} C_VEL
LIN {X 0,Y 104.84,Z 483.585,A -85,B 0,C 180,E1 -27596.593,E2 -27596.593} C_VEL
LIN {X 0,Y 104.053,Z 486.798,A -85,B 0,C 180,E1 -27597.738,E2 -27597.738} C_VEL
LIN {X 0,Y 101.696,Z 491.103,A -85,B 0,C 180,E1 -27598.863,E2 -27598.863} C_VEL
LIN {X 0,Y 96.461,Z 498.459,A -85,B 0,C 180,E1 -27600.802,E2 -27600.802} C_VEL
LIN {X 0,Y 95.269,Z 500.474,A -85,B 0,C 180,E1 -27601.62,E2 -27601.62} C_VEL
LIN {X 0,Y 90.74,Z 508.962,A -85,B 0,C 180,E1 -27606.009,E2 -27606.009} C_VEL
LIN {X 0,Y 85.755,Z 517.682,A -85,B 0,C 180,E1 -27612.103,E2 -27612.103} C_VEL
LIN {X 0,Y 81.813,Z 524.629,A -85,B 0,C 180,E1 -27618.857,E2 -27618.857} C_VEL
LIN {X 0,Y 78.652,Z 531.01,A -85,B 0,C 180,E1 -27627.44,E2 -27627.44} C_VEL
LIN {X 0,Y 76.987,Z 535.21,A -85,B 0,C 180,E1 -27635.239,E2 -27635.239} C_VEL
LIN {X 0,Y 76.36,Z 537.429,A -85,B 0,C 180,E1 -27640.608,E2 -27640.608} C_VEL
LIN {X 0,Y 76.309,Z 539.169,A -85,B 0,C 180,E1 -27646.04,E2 -27646.04} C_VEL
LIN {X 0,Y 77.544,Z 541.13,A -85,B 0,C 180,E1 -27654.999,E2 -27654.999} C_VEL
LIN {X 0,Y 79.527,Z 541.871,A -85,B 0,C 180,E1 -27662.022,E2 -27662.022} C_VEL
LIN {X 0,Y 84.098,Z 541.625,A -85,B 0,C 180,E1 -27671.227,E2 -27671.227} C_VEL
LIN {X 0,Y 87.663,Z 540.779,A -85,B 0,C 180,E1 -27676.181,E2 -27676.181} C_VEL
LIN {X 0,Y 95.149,Z 538.006,A -85,B 0,C 180,E1 -27683.78,E2 -27683.78} C_VEL
LIN {X 0,Y 102.342,Z 534.459,A -85,B 0,C 180,E1 -27689.137,E2 -27689.137} C_VEL
LIN {X 0,Y 109.899,Z 529.898,A -85,B 0,C 180,E1 -27693.545,E2 -27693.545} C_VEL
LIN {X 0,Y 118.029,Z 524.027,A -85,B 0,C 180,E1 -27697.359,E2 -27697.359} C_VEL
LIN {X 0,Y 119.723,Z 522.393,A -85,B 0,C 180,E1 -27698.478,E2 -27698.478} C_VEL
LIN {X 0,Y 121.041,Z 519.548,A -85,B 0,C 180,E1 -27701.88,E2 -27701.88} C_VEL
LIN {X 0,Y 122.151,Z 516.058,A -85,B 0,C 180,E1 -27706.695,E2 -27706.695} C_VEL
LIN {X 0,Y 122.59,Z 514.026,A -85,B 0,C 180,E1 -27710.097,E2 -27710.097} C_VEL
LIN {X 0,Y 122.929,Z 512.335,A -85,B 0,C 180,E1 -27713.435,E2 -27713.435} C_VEL
LIN {X 0,Y 123.272,Z 510.906,A -85,B 0,C 180,E1 -27716.732,E2 -27716.732} C_VEL
LIN {X 0,Y 123.531,Z 509.866,A -85,B 0,C 180,E1 -27720.001,E2 -27720.001} C_VEL
LIN {X 0,Y 123.324,Z 509.629,A -85,B 0,C 180,E1 -27723.268,E2 -27723.268} C_VEL
LIN {X 0,Y 123.08,Z 509.801,A -85,B 0,C 180,E1 -27726.558,E2 -27726.558} C_VEL
LIN {X 0,Y 122.899,Z 510.335,A -85,B 0,C 180,E1 -27729.879,E2 -27729.879} C_VEL
LIN {X 0,Y 122.756,Z 511.236,A -85,B 0,C 180,E1 -27733.277,E2 -27733.277} C_VEL
LIN {X 0,Y 122.544,Z 512.589,A -85,B 0,C 180,E1 -27736.664,E2 -27736.664} C_VEL
LIN {X 0,Y 122.271,Z 514.35,A -85,B 0,C 180,E1 -27740.175,E2 -27740.175} C_VEL
LIN {X 0,Y 121.802,Z 516.667,A -85,B 0,C 180,E1 -27743.823,E2 -27743.823} C_VEL
LIN {X 0,Y 120.669,Z 520.755,A -85,B 0,C 180,E1 -27749.118,E2 -27749.118} C_VEL
LIN {X 0,Y 119.387,Z 524.047,A -85,B 0,C 180,E1 -27752.825,E2 -27752.825} C_VEL
LIN {X 0,Y 116.641,Z 527.412,A -85,B 0,C 180,E1 -27755.569,E2 -27755.569} C_VEL
LIN {X 0,Y 114.204,Z 529.425,A -85,B 0,C 180,E1 -27756.87,E2 -27756.87} C_VEL
LIN {X 0,Y 106.563,Z 534.747,A -85,B 0,C 180,E1 -27760.673,E2 -27760.673} C_VEL
LIN {X 0,Y 99.532,Z 538.924,A -85,B 0,C 180,E1 -27765.082,E2 -27765.082} C_VEL
LIN {X 0,Y 95.221,Z 541.156,A -85,B 0,C 180,E1 -27768.374,E2 -27768.374} C_VEL
LIN {X 0,Y 91.154,Z 542.928,A -85,B 0,C 180,E1 -27771.917,E2 -27771.917} C_VEL
LIN {X 0,Y 84.38,Z 545.267,A -85,B 0,C 180,E1 -27780.017,E2 -27780.017} C_VEL
LIN {X 0,Y 81.692,Z 545.871,A -85,B 0,C 180,E1 -27784.522,E2 -27784.522} C_VEL
LIN {X 0,Y 79.658,Z 546.078,A -85,B 0,C 180,E1 -27789.334,E2 -27789.334} C_VEL
LIN {X 0,Y 77.21,Z 545.31,A -85,B 0,C 180,E1 -27799.51,E2 -27799.51} C_VEL
LIN {X 0,Y 76.85,Z 544.359,A -85,B 0,C 180,E1 -27804.752,E2 -27804.752} C_VEL
LIN {X 0,Y 76.854,Z 543.001,A -85,B 0,C 180,E1 -27809.999,E2 -27809.999} C_VEL
LIN {X 0,Y 76.946,Z 540.074,A -85,B 0,C 180,E1 -27817.873,E2 -27817.873} C_VEL
LIN {X 0,Y 78.057,Z 536.072,A -85,B 0,C 180,E1 -27825.67,E2 -27825.67} C_VEL
LIN {X 0,Y 80.831,Z 529.872,A -85,B 0,C 180,E1 -27834.392,E2 -27834.392} C_VEL
LIN {X 0,Y 84.604,Z 523.099,A -85,B 0,C 180,E1 -27841.276,E2 -27841.276} C_VEL
LIN {X 0,Y 88.891,Z 515.236,A -85,B 0,C 180,E1 -27847.229,E2 -27847.229} C_VEL
LIN {X 0,Y 93.045,Z 507.815,A -85,B 0,C 180,E1 -27851.366,E2 -27851.366} C_VEL
LIN {X 0,Y 95.519,Z 499.391,A -85,B 0,C 180,E1 -27855.836,E2 -27855.836} C_VEL
LIN {X 0,Y 97.467,Z 490.139,A -85,B 0,C 180,E1 -27860.139,E2 -27860.139} C_VEL
LIN {X 0,Y 98.499,Z 482.651,A -85,B 0,C 180,E1 -27863.33,E2 -27863.33} C_VEL
LIN {X 0,Y 97.243,Z 476.121,A -85,B 0,C 180,E1 -27867.176,E2 -27867.176} C_VEL
LIN {X 0,Y 95.893,Z 471.308,A -85,B 0,C 180,E1 -27870.349,E2 -27870.349} C_VEL
LIN {X 0,Y 93.225,Z 465.632,A -85,B 0,C 180,E1 -27875.265,E2 -27875.265} C_VEL
LIN {X 0,Y 91.444,Z 462.64,A -85,B 0,C 180,E1 -27878.588,E2 -27878.588} C_VEL
LIN {X 0,Y 90.992,Z 461.447,A -85,B 0,C 180,E1 -27879.661,E2 -27879.661} C_VEL
LIN {X 0,Y 88.868,Z 458.553,A -85,B 0,C 180,E1 -27883.93,E2 -27883.93} C_VEL
LIN {X 0,Y 88.157,Z 456.568,A -85,B 0,C 180,E1 -27886.162,E2 -27886.162} C_VEL
LIN {X 0,Y 85.955,Z 454.107,A -85,B 0,C 180,E1 -27892.068,E2 -27892.068} C_VEL
LIN {X 0,Y 85.109,Z 451.286,A -85,B 0,C 180,E1 -27897.041,E2 -27897.041} C_VEL
LIN {X 0,Y 84.349,Z 450.891,A -85,B 0,C 180,E1 -27901.105,E2 -27901.105} C_VEL
LIN {X 0,Y 84.35,Z 451.234,A -85,B 0,C 180,E1 -27914.474,E2 -27914.474} C_VEL
LIN {X 0,Y 84.71,Z 451.702,A -85,B 0,C 180,E1 -27916.88,E2 -27916.88} C_VEL
LIN {X 0,Y 86.11,Z 455.178,A -85,B 0,C 180,E1 -27924.084,E2 -27924.084} C_VEL
LIN {X 0,Y 87.902,Z 456.746,A -85,B 0,C 180,E1 -27928.666,E2 -27928.666} C_VEL
LIN {X 0,Y 89.637,Z 460.336,A -85,B 0,C 180,E1 -27933.286,E2 -27933.286} C_VEL
LIN {X 0,Y 90.808,Z 461.622,A -85,B 0,C 180,E1 -27935.482,E2 -27935.482} C_VEL
LIN {X 0,Y 93.643,Z 467.336,A -85,B 0,C 180,E1 -27941.368,E2 -27941.368} C_VEL
LIN {X 0,Y 96.029,Z 472.568,A -85,B 0,C 180,E1 -27945.957,E2 -27945.957} C_VEL
LIN {X 0,Y 98.102,Z 478.554,A -85,B 0,C 180,E1 -27950.365,E2 -27950.365} C_VEL
LIN {X 0,Y 99.144,Z 482.274,A -85,B 0,C 180,E1 -27952.889,E2 -27952.889} C_VEL
LIN {X 0,Y 98.794,Z 488.394,A -85,B 0,C 180,E1 -27955.931,E2 -27955.931} C_VEL
LIN {X 0,Y 97.925,Z 494.866,A -85,B 0,C 180,E1 -27959.247,E2 -27959.247} C_VEL
LIN {X 0,Y 95.269,Z 500.474,A -85,B 0,C 180,E1 -27961.62,E2 -27961.62} C_VEL
LIN {X 0,Y 92.512,Z 504.774,A -85,B 0,C 180,E1 -27963.445,E2 -27963.445} C_VEL
LIN {X 0,Y 86.461,Z 511.319,A -85,B 0,C 180,E1 -27966.232,E2 -27966.232} C_VEL
LIN {X 0,Y 80.342,Z 517.354,A -85,B 0,C 180,E1 -27969.69,E2 -27969.69} C_VEL
LIN {X 0,Y 77.603,Z 520.733,A -85,B 0,C 180,E1 -27972.564,E2 -27972.564} C_VEL
LIN {X 0,Y 74.286,Z 526.387,A -85,B 0,C 180,E1 -27979.094,E2 -27979.094} C_VEL
LIN {X 0,Y 71.491,Z 531.647,A -85,B 0,C 180,E1 -27987.184,E2 -27987.184} C_VEL
LIN {X 0,Y 69.768,Z 535.752,A -85,B 0,C 180,E1 -27995.782,E2 -27995.782} C_VEL
LIN {X 0,Y 69.19,Z 537.884,A -85,B 0,C 180,E1 -28001.722,E2 -28001.722} C_VEL
LIN {X 0,Y 69.314,Z 539.578,A -85,B 0,C 180,E1 -28007.71,E2 -28007.71} C_VEL
LIN {X 0,Y 70.671,Z 541.3,A -85,B 0,C 180,E1 -28016.491,E2 -28016.491} C_VEL
LIN {X 0,Y 73.334,Z 542.106,A -85,B 0,C 180,E1 -28025.101,E2 -28025.101} C_VEL
LIN {X 0,Y 78.036,Z 541.858,A -85,B 0,C 180,E1 -28033.906,E2 -28033.906} C_VEL
LIN {X 0,Y 82.672,Z 540.836,A -85,B 0,C 180,E1 -28039.915,E2 -28039.915} C_VEL
LIN {X 0,Y 90.148,Z 538.285,A -85,B 0,C 180,E1 -28046.927,E2 -28046.927} C_VEL
LIN {X 0,Y 98.729,Z 534.322,A -85,B 0,C 180,E1 -28052.849,E2 -28052.849} C_VEL
LIN {X 0,Y 106.795,Z 529.64,A -85,B 0,C 180,E1 -28057.118,E2 -28057.118} C_VEL
LIN {X 0,Y 112.478,Z 525.773,A -85,B 0,C 180,E1 -28059.593,E2 -28059.593} C_VEL
LIN {X 0,Y 114.337,Z 524.086,A -85,B 0,C 180,E1 -28061.024,E2 -28061.024} C_VEL
LIN {X 0,Y 115.466,Z 521.924,A -85,B 0,C 180,E1 -28064.106,E2 -28064.106} C_VEL
LIN {X 0,Y 116.477,Z 519.474,A -85,B 0,C 180,E1 -28068.066,E2 -28068.066} C_VEL
LIN {X 0,Y 117.237,Z 517.012,A -85,B 0,C 180,E1 -28073.115,E2 -28073.115} C_VEL
LIN {X 0,Y 117.762,Z 515.636,A -85,B 0,C 180,E1 -28076.579,E2 -28076.579} C_VEL
LIN {X 0,Y 118.151,Z 514.599,A -85,B 0,C 180,E1 -28080.001,E2 -28080.001} C_VEL
LIN {X 0,Y 118.007,Z 514.354,A -85,B 0,C 180,E1 -28083.415,E2 -28083.415} C_VEL
LIN {X 0,Y 117.725,Z 514.588,A -85,B 0,C 180,E1 -28086.858,E2 -28086.858} C_VEL
LIN {X 0,Y 117.492,Z 515.179,A -85,B 0,C 180,E1 -28090.338,E2 -28090.338} C_VEL
LIN {X 0,Y 117.077,Z 516.975,A -85,B 0,C 180,E1 -28096.167,E2 -28096.167} C_VEL
LIN {X 0,Y 116.364,Z 519.446,A -85,B 0,C 180,E1 -28101.247,E2 -28101.247} C_VEL
LIN {X 0,Y 115.48,Z 521.945,A -85,B 0,C 180,E1 -28105.216,E2 -28105.216} C_VEL
LIN {X 0,Y 114.239,Z 525.007,A -85,B 0,C 180,E1 -28109.484,E2 -28109.484} C_VEL
LIN {X 0,Y 113.28,Z 526.67,A -85,B 0,C 180,E1 -28111.454,E2 -28111.454} C_VEL
LIN {X 0,Y 112.33,Z 527.708,A -85,B 0,C 180,E1 -28112.368,E2 -28112.368} C_VEL
LIN {X 0,Y 110.097,Z 529.68,A -85,B 0,C 180,E1 -28113.918,E2 -28113.918} C_VEL
LIN {X 0,Y 102.072,Z 534.91,A -85,B 0,C 180,E1 -28117.645,E2 -28117.645} C_VEL
LIN {X 0,Y 94.639,Z 539.002,A -85,B 0,C 180,E1 -28122.046,E2 -28122.046} C_VEL
LIN {X 0,Y 90.027,Z 541.175,A -85,B 0,C 180,E1 -28125.365,E2 -28125.365} C_VEL
LIN {X 0,Y 81.78,Z 544.213,A -85,B 0,C 180,E1 -28133.018,E2 -28133.018} C_VEL
LIN {X 0,Y 75.318,Z 545.71,A -85,B 0,C 180,E1 -28142.189,E2 -28142.189} C_VEL
LIN {X 0,Y 71.349,Z 545.622,A -85,B 0,C 180,E1 -28152.811,E2 -28152.811} C_VEL
LIN {X 0,Y 69.775,Z 544.027,A -85,B 0,C 180,E1 -28164.218,E2 -28164.218} C_VEL
LIN {X 0,Y 69.752,Z 542.596,A -85,B 0,C 180,E1 -28169.999,E2 -28169.999} C_VEL
LIN {X 0,Y 69.912,Z 539.6,A -85,B 0,C 180,E1 -28178.671,E2 -28178.671} C_VEL
LIN {X 0,Y 71.214,Z 535.512,A -85,B 0,C 180,E1 -28187.22,E2 -28187.22} C_VEL
LIN {X 0,Y 74.397,Z 529.205,A -85,B 0,C 180,E1 -28196.659,E2 -28196.659} C_VEL
LIN {X 0,Y 78.551,Z 522.324,A -85,B 0,C 180,E1 -28203.998,E2 -28203.998} C_VEL
LIN {X 0,Y 82.443,Z 515.788,A -85,B 0,C 180,E1 -28209.196,E2 -28209.196} C_VEL
LIN {X 0,Y 86.759,Z 508.595,A -85,B 0,C 180,E1 -28213.51,E2 -28213.51} C_VEL
LIN {X 0,Y 89.248,Z 501.518,A -85,B 0,C 180,E1 -28217.58,E2 -28217.58} C_VEL
LIN {X 0,Y 91.42,Z 493.468,A -85,B 0,C 180,E1 -28221.698,E2 -28221.698} C_VEL
LIN {X 0,Y 92.959,Z 485.389,A -85,B 0,C 180,E1 -28225.459,E2 -28225.459} C_VEL
LIN {X 0,Y 91.843,Z 478.388,A -85,B 0,C 180,E1 -28230.171,E2 -28230.171} C_VEL
LIN {X 0,Y 90.602,Z 474.297,A -85,B 0,C 180,E1 -28233.473,E2 -28233.473} C_VEL
LIN {X 0,Y 89.142,Z 470.986,A -85,B 0,C 180,E1 -28236.783,E2 -28236.783} C_VEL
LIN {X 0,Y 87.319,Z 467.155,A -85,B 0,C 180,E1 -28241.218,E2 -28241.218} C_VEL
LIN {X 0,Y 84.905,Z 462.619,A -85,B 0,C 180,E1 -28248.056,E2 -28248.056} C_VEL
LIN {X 0,Y 82.498,Z 457.668,A -85,B 0,C 180,E1 -28259.999,E2 -28259.999} C_VEL
LIN {X 0,Y 81.847,Z 457.727,A -85,B 0,C 180,E1 -28269.888,E2 -28269.888} C_VEL
LIN {X 0,Y 82.306,Z 458.052,A -85,B 0,C 180,E1 -28274.842,E2 -28274.842} C_VEL
LIN {X 0,Y 83.024,Z 460.941,A -85,B 0,C 180,E1 -28281.39,E2 -28281.39} C_VEL
LIN {X 0,Y 84.828,Z 463.017,A -85,B 0,C 180,E1 -28287.458,E2 -28287.458} C_VEL
LIN {X 0,Y 86.188,Z 466.195,A -85,B 0,C 180,E1 -28292.006,E2 -28292.006} C_VEL
LIN {X 0,Y 87.193,Z 467.55,A -85,B 0,C 180,E1 -28294.347,E2 -28294.347} C_VEL
LIN {X 0,Y 89.528,Z 472.865,A -85,B 0,C 180,E1 -28300.333,E2 -28300.333} C_VEL
LIN {X 0,Y 91.531,Z 478.089,A -85,B 0,C 180,E1 -28305.274,E2 -28305.274} C_VEL
LIN {X 0,Y 93.326,Z 484.75,A -85,B 0,C 180,E1 -28310.522,E2 -28310.522} C_VEL
LIN {X 0,Y 93.543,Z 485.803,A -85,B 0,C 180,E1 -28311.308,E2 -28311.308} C_VEL
LIN {X 0,Y 92.362,Z 494.205,A -85,B 0,C 180,E1 -28315.865,E2 -28315.865} C_VEL
LIN {X 0,Y 91.992,Z 496.187,A -85,B 0,C 180,E1 -28317.022,E2 -28317.022} C_VEL
LIN {X 0,Y 87.214,Z 504.98,A -85,B 0,C 180,E1 -28321.087,E2 -28321.087} C_VEL
LIN {X 0,Y 82.37,Z 513.079,A -85,B 0,C 180,E1 -28326.093,E2 -28326.093} C_VEL
LIN {X 0,Y 77.603,Z 520.733,A -85,B 0,C 180,E1 -28332.564,E2 -28332.564} C_VEL
LIN {X 0,Y 75.048,Z 523.974,A -85,B 0,C 180,E1 -28335.747,E2 -28335.747} C_VEL
LIN {X 0,Y 69.697,Z 528.7,A -85,B 0,C 180,E1 -28341.202,E2 -28341.202} C_VEL
LIN {X 0,Y 64.804,Z 532.682,A -85,B 0,C 180,E1 -28347.78,E2 -28347.78} C_VEL
LIN {X 0,Y 63.116,Z 534.758,A -85,B 0,C 180,E1 -28352.542,E2 -28352.542} C_VEL
LIN {X 0,Y 62.066,Z 538.338,A -85,B 0,C 180,E1 -28363.09,E2 -28363.09} C_VEL
LIN {X 0,Y 62.372,Z 539.988,A -85,B 0,C 180,E1 -28369.758,E2 -28369.758} C_VEL
LIN {X 0,Y 63.839,Z 541.467,A -85,B 0,C 180,E1 -28378.273,E2 -28378.273} C_VEL
LIN {X 0,Y 67.388,Z 542.342,A -85,B 0,C 180,E1 -28388.738,E2 -28388.738} C_VEL
LIN {X 0,Y 72.223,Z 542.085,A -85,B 0,C 180,E1 -28397.067,E2 -28397.067} C_VEL
LIN {X 0,Y 78.089,Z 540.892,A -85,B 0,C 180,E1 -28404.095,E2 -28404.095} C_VEL
LIN {X 0,Y 85.368,Z 538.589,A -85,B 0,C 180,E1 -28410.4,E2 -28410.4} C_VEL
LIN {X 0,Y 92.834,Z 535.461,A -85,B 0,C 180,E1 -28415.293,E2 -28415.293} C_VEL
LIN {X 0,Y 101.567,Z 530.882,A -85,B 0,C 180,E1 -28419.759,E2 -28419.759} C_VEL
